(*
Nazwa:			FB_2GripperScrewers
Opis:			Zakręcarki szczekowe
Wersja:			v2.91
Data:			2026-01-12
Autor:			DP
Urzadzenia:		Serwo podnośnika, Serwo zakręcania
Ostatnie zmiany:
	- 2026-01-12 [DP] Wejście pod pozycje szukania gwintu
	- 2025-09-04 [DP] EventLog-do sprawdzenia->wywołać błędy , Estop ErrHan
	- 2025-07-09 [DP] wysokosc narzedi
	- 2025-07-08 [DP] tonError bo kasuje mcStop, tool height do błędu, opis, Resseting, Homing false w Manual
	- 2025-05-15 [DP] Zmiana errlowscrewing na -25
	- 2025-04-18 [DP] Zmiana limitu na 0.1 fullscr
	- 2025-03-31 [DP] Case 10 cofanie
	- 2025-03-31 [DP] Zmiana limitu lrPackageTurnoversToFullScrewed 0.3
	- 2025-01-17 [DP] TorqueCV 
	- 2024-12-13 [DP] Zmiany dla glowicy zasysajcej na sloiki, przejcie do pushing itd
	- 2024-12-12 [DP] Zmiana szukania gwintu
	- 2024-12-11 [DP] Skaling czuj. wysokości
	- 2024-11-26 [DP] Gear Vel sloiki
	- 2024-10-25 [DP] Zmiany torque
	- 2024-08-29 [DP] Wbijak
	- 2024-03-18 [DP] Zmiana symulacji
	- 2024-03-06 [DP] Aktualizacja instrukcji
	- 2024-02-27 [DP] Height Vel z 0 na zadaną w ressetingu, opis problemów
	- 2023-11-24 [DP] Pop. uwag dodatkowych opcji, tryb momentowy - opis
	- 2023-11-10 [DP] Akt. instrukcji, szukanie z UJL
	- 2023-03-25 [DP] przyśpieszenie screwera na stałe, zmiana instrukcji konfiguracji, skrocona czasowka griper
	- 2023-03-21 [DP] dodana ScrewerSet2
	- 2023-02-22 [DP] poprawa w GearRatio
	- 2023-02-21 [DP] Acc, Dec, Jerk i Prędkości Liftera zmniejszone 2x przez inny montaż,
				EStop w StateError, zmiana przekadni obrotu, CycleDone jak SetTorque=0,
	- 2023-02-14 [DP] Zmiana instrukcji konfiguracji
	- 2023-02-14 [DP] Wersja z LU208 z aktualizacjami z XTSa (gearing przy zakręcaniu i szukanie gwintu)
	
Konfiguracja:

Parametryzacja bloczka:
	- ustawić wysokości narzędzi, potrzebne do kolizji
	- ustawić wartość minimalną, od aktualnej wysokości zakręcarki
	

Czujnik wysokości:
	- Najlepiej przeskalować do na wejście tak, żeby pokazywał ugięcie sprężyny od transportera czyli 0mm-nieugięta
	14mm - ugięta maksymalnie (P10_GripperScrewer.IlrGripperScrewer1HeightCV:=-0.0023*(iIABPneumaticEB5AnalogueInput1)+52.006 + 1.83);

Szukanie gwintu z czujnikiem wysokości:
Włączone szukanie gwintu w pozycji dociskania i z czujnikiem wysokości, należy ustawić duży kąt obrotu (maxymalny dla szukania gwintu)
	1. Start obrotu z prędkością zadaną zakręcania, zapisywanie wartości max i min ugięcia sprężyny
	2. Szukanie 1 uskoku po 100st. o 0,5mm od wartości max ugięcia, jeżeli krotność gwintu 1x to przejście do punktu 4
	3. Szukanie 2 uskoku po 100st. jeżeli znaleziono pierwszy o 0,5mm od wartości max ugięcia
	4. Przejazd o 30,60,90st. dalej, zależnie od krotności
	5. Przejście do pozycji zakręcania lub dociskania zależnie od nastaw
	
	
Oś Obrótu (AM8031-0C20-0000): 

	Drive:
	- LU207,UBL50 - Nowa zębatka ma 32 na 48 zęby 240:360
	- ustawić driva na 'Rotatory' 360 st. i gear ratio 240:360, 240 st. na obr.
	- Invert Nc-Enc i Nc-Drive włączone
	- włączyć w drivie Scaling->Modulo data storage source - Feeback 1
	- ustawić drive Scaling->position offset setting 0 stopni na odpowiedniej pozycji na enkoderze
	- wgrać z drive Save NC parameters
	- w drivie jeszcze raz ustawić parametr Following error window 359?	
	- ustawic regulator Position mode na Kv na 10, Kp na 0.2, Tn na 0.002 
	- ustawić Acceleration Feed forward  K = 1 i wpisać inercje w Vel contr.->Vel. calc->0.001 kg m^2 oraz Mode->Basic_for_know_interia
	- ustawić w parametrach Configured channel peak current na 5A
	- ustawić w parametrach 0x6072 Bipolar torque/force limit value na 500%
	- ustawić w parametrach 0x60E0 Positive torque/force limit value na 500%
	- ustawić w parametrach 0x60E1 Negative torque/force limit value na 500%
	- dodać parametry Bipolar torque/Force limit w Process data/Outputs i polinkować ze zmienną
	- dodać parametr Positon control proportional gain Process data/Outputs i polinkować ze zmienną
	NC:
	- Ustawić Maximum Velocity na 13397.8, Reference Velocity na 14737.5, Max Acc i Dec na 300000.0
	- Default Acc i Dec na 20096.7, jerk na 60290.0
	- wyłączyć Limity Switche
	- wyłączyć wszystkie opcje Monitoringu

	Opcja trybu momentowego osi zakręcania (tylko od wersji driva 104)
	Drvie:
	- Na jednym drivie nie może być razem obrót 1 i obrót 2
	- W drivie (kanał) osi obrotu Advanced->Slots settings zaznaczyć 'I know what I do'
	i ustawiąc VelocityControlSlot na VelocityControl2, w tym momencie w IO powinny pojawić się 
	nowe wejścia,wyjścia VelocityControl2
	- W drivie Advanced->Process data rozwinąć 'Ch A Modes of operation' i ustawić '..mode_CST (10)'
	w Virual operation mode 0 
	- W parametr list powinien być parametr 0x60CA Ch a Torque limitation option code -> ustwić na
	TorqueMightBeReducedToZero, jeżeli nie ma to znaczy że trzeba zaktualizować driva lub dodać parametry ręcznie
	NC:
	- W NC w Drive->Zakładka Time Comensation-> Parametr Time Compensation Mode Drive -> 'ON(with velocity)'
	- W NC w Enc->Zakładka Time Comensation-> Parametr Time Compensation Mode Drive -> 'ON(with velocity)'
	
Oś podnoszenia (AM8032-0E21-0000):
	Drive:
	- ustawić driva na 'Linerary' 10mm i gear ratio 1:1, 10mm na obr.
	- Invert Nc-Enc i Nc-Drive włączone
	- ustawic regulator Position mode na Kv na 1, Kp na 0.2, Tn na 0.002 
	- ustawić Feed forward acceleration K = 1 i wpisać inercje w Vel contr.->Cel. calc->0 kg m^2
	NC:
	- Ustawić Maximum Velocity na 1094
	- Default Acc i Dec na 100000, jerk na 500000
	- ustawić Limit Swtiche
	- ustawić ManualVelocity (Slow) na 30 ze względu na Jog i bazowanie

Info: 
	- możliwość pracy 1 lub 2
	- możliwość pracy bez kręcenia jeżeli ustawi się prędkość 0
	- możliwosć dodatkowego chwytania przed zakręcaniem
	- step mode dla wizualizacji
	- rozróżnienie warningów

Tryb momementowy:
lrPackageTurnoversToFullScrewed - Ilośc obrotów do zakręcenia
iScrewer1SetTorque - Zadany moment w % (Przeliczany z Nm z wizualizacji)
lrScrewerSpeed - Prędkość zakręcania w st/s (Przeliczany z rpm z wizualziacji)
1. Start											Rozpędzanie,	Torque 5000 (Max) [%], 				TorqueRamp 4000 [%/s], VelocityLimitLow -5000 (Max) [st./s]
2. ActPos>lrPackageTurnoversToFullScrewed*360.0/7	Hamowanie,		Torque -9 [%],						TorqueRamp 1500 [%/s], VelocityLimitLow -4000 (Max) [st./s]
3. ActPos>lrPackageTurnoversToFullScrewed*360.0/6	Dokręcanie,		Torque iScrewer1SetTorque [%],		TorqueRamp 4000 [%/s], VelocityLimitLow lrScrewerSpeed (Max) [st./s]



Jak naprawić:
A. Zakręcarka nie wykonuje ruchu w trybie momentowym, jedna działa , druga nie - sprawdzić czy bloczek MC_Torque wykonuje ruchu,
jeżeli nie to wyłączyć VelocityControl2, włączyć bez '2' i ponownie włączyć '2', potem aktywacja
B. 
*)

FUNCTION_BLOCK FB_2GripperScrewers
VAR_INPUT
	bEnable1							:BOOL;		//Zezwolenie na pracę 1
	bEnable2							:BOOL;		//Zezwolenie na pracę 2
	bEstop								:BOOL;		//Stop awaryjny nieaktywny
	bRun1								:BOOL;		//Rozkaz zakręcania zakręcarki 1
	bRun2								:BOOL;		//Rozkaz zakręcania zakręcarki 2
	bSimulation							:BOOL;		//Włączona symulacja, skracanie czasu przerywania jak nie ma butelki
	bHoming								:BOOL;		//Zezwolenie na wykonanie bazowania i pozycjonowania zakręcarki
	bHeightSet							:BOOL;		//Ustaw wysokość
	bIgnoreError						:BOOL;		//Ignorowania błędów cyklu pracy
	bScrewer1SetPositionOffset			:BOOL;		//Ustaw offset obrotu zakręcarki 1
	bScrewer2SetPositionOffset			:BOOL;		//Ustaw offset obrotu zakręcarki 2
	iScrewer1AddTorque					:UINT;
	iScrewer2AddTorque					:UINT;
	bReset								:BOOL;		//Reset błędu, jeśli w stanie "eError
	iTool								:INT;		// Wybór narzędzia (1-5), opisy w tablicy AsGripperScrewerTool	
	bOptionOpenedGripperWhenFindingScrew:BOOL;		//OPCJA. Otwarty chwytak przy szukaniu gwintu
	bOptionScrewingBackwardsInPushingPosition:BOOL;	//OPCJA. Obrót do tyłu w pozycji dociskania
	bOptionCapPushingWithoutScrewing	:BOOL;		//OPCJA. Tylko wbijanie bez zakręcania
	bOptionCapPositioning				:BOOL;		//OPCJA. Dodatkowe zamknięcie chwytakiem przed zakręceniem (do testów)
	bOptionFindScrewInScrewingPosition	:BOOL;		//OPCJA. Szukaj początku gwintu nakrętki i opakowania. Zakręcarka napjpierw obraca się w lewo, a po znalezienu gwintu przystepuje do zakręcania w pozycji zakręcania
	bOptionFindScrewInPushingPosition	:BOOL;		//OPCJA. Szukaj początku gwintu nakrętki i opakowania. Zakręcarka napjpierw obraca się w lewo, a po znalezienu gwintu przystepuje do zakręcania w pozycsji docisku
	bOptionFindScrewWithHeightSensor	:BOOL;		//OPCJA. Szukanie gwintu z czujnikiem wysokości
	bOptionFindScrewRotateFromPushingToScrewingSensor	:BOOL;		//OPCJA. Obrót od pozycji docisku do zakręcania
	bOptionMomentaryMode				:BOOL;		//OPCJA. Tryb momentowy zakręcania
	lrPackageTurnoversToFullScrewed		:LREAL;		//Obroty do pełnego zakręcenia
	lrPackageThreadPitch				:LREAL;		//Skok gwintu
	lrPackageThreadTimes				:LREAL;		//Krotność gwintu
	lrHeightReadyPosition				:LREAL;		//Wysokość zadana w stanie gotowości od płyty[mm]
	lrHeightPushingPosition				:LREAL;		//Wysokość zadana przy wciskaniu nakrętki od płyty[mm]
	lrHeightEndScrewingPosition			:LREAL;		//Wysokość zadana przy zakręcaniu nakrętki od płyty [mm]
	lrHeightFindScrewPosition			:LREAL;		//Pozycja szukania gwintu [mm]
	lrHeightScrewingDistanceSpeed		:REAL;		//Prędkość obniżania podczas zakręcania
	lrHeightActualPosition				:LREAL;		//Aktualna pozycja podnośnika
	lrSpringHeightCV					:LREAL;		//Czujnik ugięcia sprężyny (przeskalować na 0-14mm (14mm-maksymalnie ugięta)
	lrHeightActualTorque				:LREAL;		//Aktualny moment [%]
	rActualMotor1Temperature			:REAL;		//Aktualna temperatura silnika 1
	rActualMotor2Temperature			:REAL;		//Aktualna temperatura silnika 2
	iHeightSetTorque					:INT;		//Zadany moment dociskania [%]
	iScrewer1SetTorque					:INT;		//Zadany moment dokręcania [%]
	iScrewer2SetTorque					:INT;		//Zadany moment dokręcania [%]
	iScrewTightTime						:INT;		//Czas przytrzymania po uzyskaniu momentu [ms] 
	lrScrewer1ActualTorque				:LREAL;		//Aktualny moment [%]
	lrScrewer2ActualTorque				:LREAL;		//Aktualny moment [%]
	lrHeightAcceleration				:LREAL;		//Przyspieszenie podnosnika zakręcarki
	lrHeightDeceleration				:LREAL;		//Opóźnienie podnośnika zakręcarki
	lrHeightSpeed						:LREAL;		//Prędkość podnośnika zakręcarki
	lrScrewer1ActualPosition			:LREAL;	
	lrScrewer2ActualPosition			:LREAL;	
	lrScrewerAcceleration				:LREAL;		//Przyspieszenie zakręcania
	lrScrewerDeceleration				:LREAL;		//Opóźnienie zakręcania
	lrScrewerSpeed						:LREAL;		//Prędkość zakręcania
	lrScrewer1PosDiff					:LREAL;		//ScrewingAxisRef.NcToPlc.PosDiff
	lrScrewer2PosDiff					:LREAL;		//ScrewingAxisRef.NcToPlc.PosDiff
	lrFindigScrewDegree					:LREAL;		//Kąt wycofania zakręcarki przy szukaniu gwintu
	bManualMovement						:BOOL;		//Zezwolenie na ruchy ręcznę
	lrManualOverride					:LREAL;		//Procentowa redukcja prędkości wszystkich serw (Tylko w trybie manualnym)
                                	
	lrMaxHeightPosition:LREAL;				//Wysokość maksymalna zakręcarki 
	lrMinHeightPosition:LREAL;				//Wysokość minimalna zakręcarki 
	lrMaxScrewerSpeed	:LREAL;				//Maksymalna prędkość zakręcania

	//StepMode
	bStepMode				: BOOL;		//Włączony tryb skokowy sterowania podnośnikami (tylko w serwisie)
	lrSetPosStepMode		: LREAL; 	//Ruch podnośnika o zadaną wartość w trybie krokowym (tylko w serwisie)
	
	_ALARMINFO_ :BOOL;
	iStationIndex:UDINT;					//Numer stacji 
	sStationName:WSTRING;					//Nazwa stacji
END_VAR

VAR_OUTPUT
	eState							: E_Station;				//Stan ogólny bloku
	eRunningState					: E_GripperScrewer; 		//Stan zakręcarki
	bError							: BOOL;						//Błąd stacji
	udiErrorID						: UDINT;					//Nr błędu zakręcarki
	sErrorDescription				: STRING(200);				//Opis błędu
	sErrorDescription2				: STRING(200);				//Opis błędu
	sErrorStationName				: STRING;					//Nazwa stacj
	udiStationID					: UDINT;				// Nr stacji
	
	udiHeightServoErrorNr			: UDINT;					//Nr błędu serwo podnośnika
	udiScrewing1ServoErrorNr		: UDINT;					//Nr błędu serwo zakręcarki 1
	udiScrewing2ServoErrorNr		: UDINT;					//Nr błędu serwo zakręcarki 2
	bGripper1Actuator				: BOOL;						//Siłownik chwytaka
	bGripper2Actuator				: BOOL;						//Siłownik chwytaka
	uiScrewing1TorqueControl		: UINT;						//Kontola momentu zakręcania	
	uiScrewing2TorqueControl		: UINT;						//Kontola momentu zakręcania	
	rScrewing1ProportionalGain		: UINT;						//Kontola Kp
	rScrewing2ProportionalGain		: UINT;						//Kontola Kp	
	lrScrewer1TorqueCV				: LREAL;					//Wartość osiągniętego momentu dokręcenia [nM]
	lrScrewer2TorqueCV				: LREAL;					//Wartość osiągniętego momentu dokręcenia [nM]
	uiHeightTorqueControl			: UINT						:= 6000;
	sWarningDescription				: STRING;
	bWarning1						: BOOL;
	bWarning1A						: BOOL;	
	bWarning1B						: BOOL;	
	bWarning1C						: BOOL;	
	bWarning1D						: BOOL;	
	bWarning1E						: BOOL;	{warning'dorobic ostrzezenie szukania gwintu}
	bWarning2						: BOOL;
	bWarning2A						: BOOL;	
	bWarning2B						: BOOL;	
	bWarning2C						: BOOL;	
	bWarning2D						: BOOL;	
	bWarning2E						: BOOL;	
	udiWarningID					: UDINT;
	tCycleTime						: TIME;	
	bHomingDone						: BOOL;						//Wymagane ponowne bazowanie (blad podczas bazowania lub stop awaryjny)
	bCycleDone1						: BOOL;
	bCycleNotDone1					: BOOL;		
	bCycleDone2						: BOOL;
	bCycleNotDone2					: BOOL;		
	bAdjustingTorqueDone			: BOOL;
	iAdjustingTorque				: INT;
	lrAdjustingMaxTorque			: LREAL;
	AsToolDescription				: ARRAY [0..10] OF STRING;	// Opis narzędzi, 1 - Opis narzędzia nr 1, 2 - Opis narzędzia nr 2
	sTool							: STRING;
	iToolHeight						: INT;	//Wysokość narzędzia od dolnej metalowej częsci dwuszczekowego
END_VAR

VAR_IN_OUT
	bManualHeightUp					:BOOL;			//Ruch ręczny podnośnikiem stacji w górę
	bManualHeightDown				:BOOL;			//Ruch ręczny podnośnikiem stacji w dół
	bManualScrew1Clockwise			:BOOL;			//Ruch ręczny zakręcarką w kierunku wskazówek zegara;
	bManualScrew1CClockwise			:BOOL;			//Ruch ręczny zakręcarką w kierunku przeciwnym do wskazówek zegara;
	bManualScrew2Clockwise			:BOOL;			//Ruch ręczny zakręcarką w kierunku wskazówek zegara;
	bManualScrew2CClockwise			:BOOL;			//Ruch ręczny zakręcarką w kierunku przeciwnym do wskazówek zegara;
	bManualGripper1					:BOOL;			//Ruch zamknięcie chwytaka nakrętek
	bManualGripper2					:BOOL;			//Ruch zamknięcie chwytaka nakrętek
	HeightAxisRef					:AXIS_REF;		//Struktura sterowania NC dla serwa podnoszenia zakręcarki
	Screwing1AxisRef				:AXIS_REF;		//Struktura sterowania NC dla serwa zakręcania
	Screwing2AxisRef				:AXIS_REF;		//Struktura sterowania NC dla serwa zakręcania	
	bFindScrewAdjustSensorHeight	:BOOL;			//Włacz szukanie MIN i MAX jeżeli jest opcja z czujnikie wysokości
	bAdjustingTorque				:BOOL;			//Dobieranie momentu
	lrAdjustingSetTorque			:LREAL;	
END_VAR

VAR
	bScrew1Found					: BOOL; 						// Zakręcarka znalazła początek gwintu
	bScrew2Found					: BOOL; 						// Zakręcarka znalazła początek gwintu	
	tonTightScrewing1Timer			: TON; 							// Timer potwierdzenia dokręcenia nakrętki
	tonTightScrewing2Timer			: TON; 							// Timer potwierdzenia dokręcenia nakrętki
	tonTightScrewing1TimerAndOpenedGripper	: TON; 					// Timer potwierdzenia dokręcenia nakrętki
	tonTightScrewing2TimerAndOpenedGripper	: TON; 					// Timer potwierdzenia dokręcenia nakrętki	
	tonMomentaryScrewing1Timer		: TON; 							// Timer potwierdzenia dokręcenia nakrętki
	tonMomentaryScrewing2Timer		: TON; 							// Timer potwierdzenia dokręcenia nakrętki

	bScrewed1					: BOOL; 						// Nakrętka zakręcona
	bScrewed2					: BOOL; 						// Nakrętka zakręcona
	tonTooLongScrewing1			: TON;							// Błąd zbyt długiego zakręcania
	tonTooLongScrewing2			: TON; 							// Błąd zbyt długiego zakręcania	
	tTooLongScrewing1			: TIME;							// Czas  zbyt długiego zakręcania
	tTooLongScrewing2			: TIME; 						// Czas  zbyt długiego zakręcania		
	tonGripper1ReliseDelay		: TON;							// Time Opóźniajacy ruch w górę po zakręceniu, pozwalajac na otwarcie chwytaka
	tonGripper2ReliseDelay		: TON;							// Time Opóźniajacy ruch w górę po zakręceniu, pozwalajac na otwarcie chwytaka
	tonGripper1ReliseDelay2		: TON;							// Time Opóźniajacy ruch w górę po zakręceniu, pozwalajac na otwarcie chwytaka
	tonGripper2ReliseDelay2		: TON;							// Time Opóźniajacy ruch w górę po zakręceniu, pozwalajac na otwarcie chwytaka

	mcScrewer1ManualMove		: MC_JOG; 						// Blok obrotu ręcznego zakręcarką
	mcScrewer2ManualMove		: MC_JOG; 						// Blok obrotu ręcznego zakręcarką
	mcScrewer1Stop				: MC_Stop;						// Trwałe zatrzymywanie Serwo
	mcScrewer2Stop				: MC_Stop;						// Trwałe zatrzymywanie Serwo
	mcScrewer1MoveVelocity		: MC_MoveVelocity;				// Ruch prędkościowy
	mcScrewer2MoveVelocity		: MC_MoveVelocity;				// Ruch prędkościowy
	mcScrewer1MoveVelocity2		: MC_MoveVelocity;				// Ruch prędkościowy
	mcScrewer2MoveVelocity2		: MC_MoveVelocity;				// Ruch prędkościowy
	mcScrewer1MoveVelocity3		: MC_MoveVelocity;				// Ruch prędkościowy
	mcScrewer2MoveVelocity3		: MC_MoveVelocity;				// Ruch prędkościowy	
	mcScrewer1MoveRelative		: MC_MoveRelative; 				// Ruch relatywny zakręcarki
	mcScrewer2MoveRelative		: MC_MoveRelative; 				// Ruch relatywny zakręcarki
	mcScrewer1MoveAbsolute		: MC_MoveAbsolute; 				// Ruch absolutny zakręcarki
	mcScrewer2MoveAbsolute		: MC_MoveAbsolute; 				// Ruch absolutny zakręcarki
	fbScrewer1SetPositionOffset	: FB_CoEAX8000SetPositionOffset;// Ustawianie pozycji obrotu 
	fbScrewer2SetPositionOffset	: FB_CoEAX8000SetPositionOffset;// Ustawianie pozycji obrotu 
	mcScrewer1TorqueControl		: MC_TorqueControl;
	mcScrewer2TorqueControl		: MC_TorqueControl;
	
	mcScrewing1Power			: MC_Power;			 			// Zasilanie napędu zakręcarki
	mcScrewing2Power			: MC_Power;			 			// Zasilanie napędu zakręcarki
	bScrewer1ServoPower			: BOOL; 						// Zmienna sterujaca zasilaniem serwo Zakręcarki
	bScrewer2ServoPower			: BOOL; 						// Zmienna sterujaca zasilaniem serwo Zakręcarki
	fbScrewer1HardReset			: FB_SoEReset; 					// Blok twardego resetu serwa zakręcania
	fbScrewer2HardReset			: FB_SoEReset; 					// Blok twardego resetu serwa zakręcania
	mcScrewer1SoftReset			: MC_Reset; 					// blok łagodnego resetu serwa zakręcarki
	mcScrewer2SoftReset			: MC_Reset; 					// blok łagodnego resetu serwa zakręcarki
	
	mcHeightManualMove			: MC_JOG; 						// Blok sterowania ręcznego wysokością
	mcHeightStop				: MC_STOP; 						// Trwałe Zatrzymywanie ruchu podnośnika zakręcarki
	mcHeightMoveAbsolute		: MC_MoveAbsolute;				// Blok sterowania wysokością	
	mcHeightPower				: MC_POWER; 					// Uruchomienie zasilania serwa podnosnika zakręcarki
	bHeightServoPower			: BOOL; 						// Zmienna sterowania zasilaniem serwo
	fbHeightHardReset			: FB_SoEReset; 					// Blok Twardego resetu serwa podnośnika zakręcarki
	mcHeightSoftReset			: MC_Reset; 					// Blok łagonego resetu podnośnika zakręcarki
	mcHeightGearInMultiMaster	: MC_GearInMultiMaster; 		// Blok sprzęgania podnoszenia z zakręcaniem
	mcHeightGearOut				: Mc_GearOut;					// Blok wysprzeglania podnoszenia z zakręcaniem

	(*Axis online*)
	fbHeight					: FB_McAxisOnlineAX8000;
	stHeight					: ST_McAxisOnline;
	fbScrewing1					: FB_McAxisOnlineAX8000;
	stScrewing1					: ST_McAxisOnline;
	fbScrewing2					: FB_McAxisOnlineAX8000;
	stScrewing2					: ST_McAxisOnline;
	
	(*Ostrzezenia,przerywanie*)
	tonTooLongFinding1			: TON; 							// Za długie szukanie gwintu
	tonTooLongFinding2			: TON; 							// Za długie szukanie gwintu
	tonPosDiff1Error			: TON;
	tonPosDiff2Error			: TON;
	tonPosTooLowWhenScrewing1	: TON;
	tonPosTooLowWhenScrewing2	: TON;
	
	(*Statistics*)
	tonCycleTimer				: TON;
	rtrigCycleTimerRead			: R_TRIG;

	lrStartPosition1			: LREAL;
	lrStartPosition2			: LREAL;
	tonMaxHeight				: TON;

	tonGripper1Delay			: TON;
	tonGripper2Delay			: TON;
	
	eLastState					: E_Station;			// Stan ogólny bloku
	eLastRunningState			: E_GripperScrewer;		// Stan podbloku
	eLastStateTemp				: E_Station;			// Stan ogólny bloku
	eLastRunningStateTemp		: E_GripperScrewer;		// Stan podbloku

	bStateError: BOOL;
	bHeighSetNotDone: BOOL;
	
	(*Szukanie momentu*)
	nCaseAdjustingTorque					: INT;
	tonAdjustingTightScrewingTimer			: TON;
	tonAdjustingGripperClose				: TON;
	uiAdjustingScrewerTorqueControl			: UINT;
	bAdjustingScrewed						: BOOL;
	tonAdjustingCase40						: TON;
	bAdjustingSetTorqueAchieved				: BOOL;
	bAdjustingTorqueTooHigh					: BOOL;
	bAdjustingTorqueTooLow					: BOOL;
	lrMotorNominalTorque					: LREAL;
	lrScrewerActualTorqueNm					: LREAL;
	
	tonFindingScrew						: TON;
	tonScrew1Found						: TON;
	tonScrew2Found						: TON;
	tonDelayServoOn						: TON;

	bPreparingToDisable					: BOOL;
	bHeightGearingWithScrewer			: BOOL;
	iStoppingCase						: INT;
	iScrewingCase						: INT;
	iScrewing2Case						: INT;
	
	(*Bledy, Resetowanie*)
	tonResetting						: TON;
	tonEstop							: TON;
	tonError							: TON;	
	rtResetCommands						: R_TRIG;
	tonActualMotor1TemperatureTooHigh	: TON;
	tonActualMotor2TemperatureTooHigh	: TON;
	iErrorResseting3					: INT;
	iTestError3							: INT;
	iTestError4							: INT;
	
	(*Metoda*)
	mcMoveAbsolute						: MC_MoveAbsolute; 				// Ruch absolutny
	iMStep								: INT;							// Do testów
	bPrepareToReadyTest					: BOOL;							// Do testów	

	(*Bazowanie*)
	iHomingCase							: INT;
	iPreparingToReadyCase				: INT;
	
	(*Czytanie momentu*)
	rtRun1								: R_TRIG;
	rtRun2								: R_TRIG;

	(*Step Mode*)
	rtStepModeUp						: R_TRIG;
	rtStepModeDown						: R_TRIG;
	lrStepModeHeightMotorSV				: LREAL;
	bStepModeMoving						: BOOL;
	tofStepModeMoving					: TOF;	
	
	(*Running*)
	iGoingUpCase						: INT;
	iToPushingPositionCase				: INT;
	tonDelayBeforeResetLag				: TON;
	lrGearRatio1						: LREAL;
	lrGearRatio2						: LREAL;
	lrSf1								: LREAL;	
	lrSf2								: LREAL;
	lrDivider							: LREAL;	
	
	(*Dodatkowe chwytanie przed zakreceniem*)
	iCloseGripperBeforeScrewingCASE		: INT;
	
	(*Bez zakręcania*)
	tonHoldingTimer						: TON;
	
	(*Aborting*)
	iAbortingCASE						: INT;
	
	(*Szukanie gwintu*)
	iFindingScrewCASE							: INT;
	lrScrewer1MaxTorqueWhenFindingScrew			: LREAL; //OPCJA 1
	lrScrewer2MaxTorqueWhenFindingScrew			: LREAL; //OPCJA 1	
	lrScrewerMinTorqueWhenFindingScrew			: LREAL; //OPCJA 1
	lrScrewerMaxSensorHeightWhenFindingScrew	: LREAL:= -100000; //OPCJA 2
	lrScrewerMinSensorHeightWhenFindingScrew	: LREAL:= 0; //OPCJA 2
	bScrew1MinFound								: BOOL;
	bScrew2MinFound								: BOOL;
	lrStartPosition1FindingScrew				: LREAL;
	lrStartPosition2FindingScrew				: LREAL;
	lrFindingScrewPositionDelay					: LREAL;	
	tonFindingScrewDelay						: TON;
	iFindScrewAdjustSensorHeight				: INT;
	
	(*Symulacja*)
	tonSimulationScrewing1						: TON;
	tonSimulationScrewing2						: TON;	
	
	(*inne*)
	iTestResetting: INT;
	iCountAborting: INT;
	bTest2:BOOL;
	lrScrewerOffsetSensorHeightWhenFindingScrew: LREAL;
	bTest: BOOL;
	iTesty: INT;
	tonTesty1: TON;
	tonTesty2: TON;	
	
	//Zmienne od EVENTLOGGER
	bAlarmInit 						: BOOL := TRUE; 
	nAlarmNumerator					: INT;
	arfbAlarm						: ARRAY[0..19] OF  FB_TcAlarm;		//Tablica bloczków błędów
	fbSourceInfo 					: FB_TcSourceInfo;
	iSourceInfo						: I_TcSourceInfo;
	sAlarmTest						: STRING;
	//Koniec zmiennych od EVENTLOGGER
	
END_VAR

IF bPrepareToReadyTest THEN
	IF	M_PrepareToReady(	AxisRef			:=  Screwing1AxisRef,			
                   			iGripperArms	:=	2
						)	
	THEN
		bPrepareToReadyTest := FALSE;
	END_IF			
				   
END_IF  

//Wywołanie AXIS Online
(*fbHeight	(stMcAxisOnline:= stHeight,		Axis:= HeightAxisRef);
fbHeight	(stMcAxisOnline:= stHeight,		Axis:= HeightAxisRef);
fbScrewing1	(stMcAxisOnline:= stScrewing1,	Axis:= Screwing1AxisRef);
fbScrewing1	(stMcAxisOnline:= stScrewing1,	Axis:= Screwing1AxisRef);
fbScrewing2	(stMcAxisOnline:= stScrewing2,	Axis:= Screwing2AxisRef);
fbScrewing2	(stMcAxisOnline:= stScrewing2,	Axis:= Screwing2AxisRef);
*)
//Parametryzacja
bHeightGearingWithScrewer := TRUE;

Tools();
ErrorHandling();
Control();
Limits();
AdjustingTorque();
HeightControlBlocks();
TorqueControl();
Screwer1ControlBlocks();
Screwer2ControlBlocks();
Simulation();
ReadScrewingTorque();
Statistics();
Warnings();
aStationID();
aTesty();
(*Zapisywanie ostatniego stanu*)
IF eLastStateTemp<>eState THEN
	eLastState := eLastStateTemp;
END_IF
eLastStateTemp := eState;
IF eLastRunningStateTemp<>eRunningState THEN
	eLastRunningState := eLastRunningStateTemp;
END_IF
eLastRunningStateTemp := eRunningState;
(*Koniec Zapisywanie ostatniego stanu*)


(*Dodatkowe zabezpieczenie przed uderzeniem w chwytak*)
IF mcHeightMoveAbsolute.Execute AND (mcHeightMoveAbsolute.Position-iToolHeight)<=lrMinHeightPosition THEN
	mcHeightMoveAbsolute.Execute:=FALSE;
END_IF
	
IF mcHeightMoveAbsolute.Error THEN
	mcHeightMoveAbsolute.Execute:=FALSE;
END_IF

IF mcScrewer1MoveVelocity.Error THEN
	mcScrewer1MoveVelocity.Execute:=FALSE;
END_IF	
(*Koniec dodatkowe zabezpieczenie przed uderzeniem w chwytak*)


(*Zabezpieczenie przed kolizją stacji poprzez ruch podnośnika*)	
IF bManualHeightDown AND (HeightAxisRef.NcToPlc.ActPos-iToolHeight)<=lrMinHeightPosition AND NOT bHoming AND NOT bHeightSet THEN
	bManualHeightDown:=FALSE;
END_IF	

IF bManualHeightUp AND (HeightAxisRef.NcToPlc.ActPos)>=lrMaxHeightPosition AND NOT bHoming AND NOT bHeightSet THEN
	bManualHeightUp:=FALSE;
END_IF	
(*Koniec zabezpieczenia przed kolizją stacji poprzez ruch podnośnika*)

ACTION AdjustingTorque:
(*

bAdjustingTorque;								// Wlączenie szukania 
lrAdjustingSetTorque;							// Szukany moment [Nm]
uiAdjustingScrewerTorqueControl; 				// Badanie tym momentem, zwiekszanie o ileś
lrMotorNominalTorque					:=	3.192; 		

tonAdjustingGripperClose		(IN:=	bGripper1Actuator, 																		PT:=T#200MS);
tonAdjustingTightScrewingTimer	(IN:=	nCaseAdjustingTorque = 30 AND (lrScrewer1ActualTorque>=uiAdjustingScrewerTorqueControl),	PT:=T#1000MS);
tonAdjustingCase40				(IN:=	nCaseAdjustingTorque=40,																PT:=T#200MS);

CASE nCaseAdjustingTorque OF
	
	0: //Włączanie
		IF bAdjustingTorque AND NOT bAdjustingTorqueDone THEN
			//Kasowanie zmiennych
			lrStartPosition1				:=	0;
			uiAdjustingScrewerTorqueControl	:=	0;
			iAdjustingTorque				:=  0;
			lrAdjustingMaxTorque			:= 	0;
			bAdjustingTorqueTooHigh			:=	FALSE;
			bAdjustingTorqueTooLow			:=	FALSE;
			nCaseAdjustingTorque			:=	10;
			mcScrewer1MoveVelocity.Execute	:=	FALSE;
		END_IF
		
	10: //Zamykanie chwytaka
		bGripper1Actuator					:=	TRUE;
		IF tonAdjustingGripperClose.Q THEN
			nCaseAdjustingTorque			:=	20;
		END_IF
		
	20:	//Ustawienie dużego momentu na początek ruchu
		uiScrewing1TorqueControl				:=  6000;
		lrStartPosition1						:=	Screwing1AxisRef.NcToPlc.ActPos;		

		IF  bAdjustingTorqueTooLow	THEN
			bAdjustingTorqueTooLow				:= FALSE;
			uiAdjustingScrewerTorqueControl		:=  uiAdjustingScrewerTorqueControl + 1;
		ELSIF bAdjustingTorqueTooHigh	THEN
			bAdjustingTorqueTooHigh				:= FALSE;
			IF uiAdjustingScrewerTorqueControl	>	0 THEN
			uiAdjustingScrewerTorqueControl		:=  uiAdjustingScrewerTorqueControl - 1;
			END_IF
		END_IF
		nCaseAdjustingTorque				:=	30;
		
	30:	 //Zakręcanie

		//Zacznij zakręcać
		lrScrewerAcceleration				:=	26000;
		lrScrewerDeceleration				:=	26000;
		mcScrewer1MoveVelocity.Direction		:=	MC_Positive_Direction;
		mcScrewer1MoveVelocity.Velocity		:=	5000;
		mcScrewer1MoveVelocity.Execute		:=	TRUE;
		
		//Zwiększanie momentu na początek ruchu
		IF ABS(ABS(lrStartPosition1)-ABS(Screwing1AxisRef.NcToPlc.ActPos))>15 OR ABS(Screwing1AxisRef.NcToPlc.PosDiff)>15  THEN 
			uiScrewing1TorqueControl			:=	(uiAdjustingScrewerTorqueControl+3)*10;
		ELSE
			uiScrewing1TorqueControl			:=	(uiAdjustingScrewerTorqueControl+3)*10+500;	
		END_IF
		
		IF tonAdjustingTightScrewingTimer.Q THEN //Jeżeli osiągnięty moment przez 200MS
			mcScrewer1MoveVelocity.Execute	:=	FALSE;
			mcScrewer1SoftReset				(Axis:=Screwing1AxisRef, Execute:= TRUE);
			iAdjustingTorque				:= UINT_TO_INT(uiScrewing1TorqueControl/10);
			uiScrewing1TorqueControl			:=	0;
			bAdjustingScrewed				:=	TRUE;		
		END_IF
			   
		IF mcScrewer1MoveVelocity.Execute = FALSE AND bAdjustingScrewed THEN
			nCaseAdjustingTorque			:=	40;
		
		END_IF	
		
	40:	//Czekanie po zakręceniu
		mcScrewer1SoftReset					(Axis:=Screwing1AxisRef, Execute:= FALSE);
		uiScrewing1TorqueControl				:=	0;
		lrStartPosition1						:=	0;
		lrAdjustingMaxTorque				:= 	0;
		bAdjustingScrewed					:=	FALSE;
		IF tonAdjustingCase40.Q THEN
			lrStartPosition1					:=	Screwing1AxisRef.NcToPlc.ActPos;	
			uiScrewing1TorqueControl			:=	1;
			nCaseAdjustingTorque			:=	50;
		END_IF
		
	50: //Odkręcanie

		lrScrewerAcceleration				:=	20;
		lrScrewerDeceleration				:=	20;
		mcScrewer1MoveVelocity.Direction		:=	MC_Negative_Direction;
		mcScrewer1MoveVelocity.Velocity		:=	10;
		mcScrewer1MoveVelocity.Execute		:=	TRUE;
		uiScrewing1TorqueControl				:=	6000;
		
		//Szukanie największego momentu w Nm
		lrScrewerActualTorqueNm:=(ABS(lrScrewer1ActualTorque)/100.0)*lrMotorNominalTorque;
		IF lrScrewerActualTorqueNm	>=	lrAdjustingMaxTorque THEN
			lrAdjustingMaxTorque			:=	lrScrewerActualTorqueNm;
		END_IF
		
		//Jeżeli osiągnięty moment
		IF lrAdjustingMaxTorque>=lrAdjustingSetTorque - 0.1 AND lrAdjustingMaxTorque<=lrAdjustingSetTorque + 0.1 THEN
			bAdjustingSetTorqueAchieved 	:= TRUE;
		ELSE
			bAdjustingSetTorqueAchieved 	:= FALSE;
		END_IF
		
		
		//Odkręcone ale nie z zadanym momentem
		IF ABS(Screwing1AxisRef.NcToPlc.ActPos-lrStartPosition1) > 45 OR ABS(Screwing1AxisRef.NcToPlc.PosDiff) > 45  THEN
			mcScrewer1SoftReset				(Axis:=Screwing1AxisRef, Execute:= TRUE);
			mcScrewer1MoveVelocity.Execute	:=	FALSE;
			
			IF lrAdjustingMaxTorque >= lrAdjustingSetTorque + 0.1 THEN
				bAdjustingTorqueTooHigh		:= TRUE;
			ELSIF lrAdjustingMaxTorque <= lrAdjustingSetTorque - 0.1 THEN
				bAdjustingTorqueTooLow		:= TRUE;	
			END_IF				
			nCaseAdjustingTorque			:= 60;
			
		END_IF
		
		//Pozycja aktualna jest większa niż 1/4 obrotu
		IF bAdjustingSetTorqueAchieved AND ABS(Screwing1AxisRef.NcToPlc.ActPos-lrStartPosition1)>45 THEN
			mcScrewer1SoftReset				(Axis:=Screwing1AxisRef, Execute:= TRUE);
			mcScrewer1MoveVelocity.Execute	:=	FALSE;
			nCaseAdjustingTorque			:= 100;
		END_IF
		
		
	60: //Ponowne zwiększanie momentu
	
		mcScrewer1SoftReset					(Axis:=Screwing1AxisRef, Execute:= FALSE);
		bAdjustingSetTorqueAchieved 		:=	FALSE;
		nCaseAdjustingTorque				:= 20;	



		
	100: //Moment znaleziony
		
		iAdjustingTorque;
		bGripper1Actuator					:= FALSE;
		nCaseAdjustingTorque				:= 0;
		//bAdjustingTorque 					:= FALSE;
		mcScrewer1MoveVelocity.Direction		:=	MC_Positive_Direction;	
		bAdjustingTorqueDone				:= TRUE;
	
END_CASE

//Resetowanie gdy wyłączono w trakcie
IF nCaseAdjustingTorque > 0 AND NOT bAdjustingTorque THEN

		lrStartPosition1					:=	0;
		uiAdjustingScrewerTorqueControl	:=	0;
		iAdjustingTorque				:=  0;
		lrAdjustingMaxTorque			:= 	0;
		bAdjustingTorqueTooHigh			:=	FALSE;
		bAdjustingTorqueTooLow			:=	FALSE;
		bAdjustingTorqueDone			:= FALSE;
		mcScrewer1Stop.Execute			:=	TRUE;
		IF mcScrewer1Stop.Done THEN
					mcScrewer1Stop.Execute			:=	FALSE;
					nCaseAdjustingTorque			:=	0;
		END_IF
END_IF

//Kasowanie Done
IF NOT bAdjustingTorque THEN 
				bAdjustingTorqueDone			:= FALSE;
END_IF
*)
END_ACTION

ACTION aStationID:
udiStationID	:=	iStationIndex;
END_ACTION

ACTION aTesty:
mcHeightMoveAbsolute;
tonTesty1	(IN:=iTesty=30, PT:=T#100MS);
tonTesty2	(IN:=iTesty=60, PT:=T#1000MS);

CASE iTesty OF 
	
		0:
			;
			
		10: 
		
			mcHeightMoveAbsolute.Execute						:=	TRUE;
			mcHeightMoveAbsolute.Velocity						:=	lrHeightSpeed;
			mcHeightMoveAbsolute.Position						:=	300;
			IF mcHeightMoveAbsolute.Done THEN
				mcHeightMoveAbsolute.Execute					:= FALSE;
				iTesty	:=	iTesty	+	10;
			END_IF
			
		20:
			mcHeightMoveAbsolute.Execute						:=	TRUE;
			mcHeightMoveAbsolute.Velocity						:=	lrHeightSpeed;
			mcHeightMoveAbsolute.Position						:=	250;
			IF mcHeightMoveAbsolute.Done THEN
				mcHeightMoveAbsolute.Execute					:= FALSE;
				iTesty	:=	iTesty	+	10;
			END_IF
			
		30:
			IF tonTesty1.Q THEN
				iTesty	:=	iTesty	+	10;
			END_IF
		
		40:
		
			mcHeightMoveAbsolute.Execute						:=	TRUE;
			mcHeightMoveAbsolute.Velocity						:=	lrHeightSpeed;
			mcHeightMoveAbsolute.Position						:=	300;
			IF mcHeightMoveAbsolute.Done THEN
				mcHeightMoveAbsolute.Execute					:= FALSE;
				iTesty	:=	iTesty	+	10;
			END_IF

		50:
		
			mcHeightMoveAbsolute.Execute						:=	TRUE;
			mcHeightMoveAbsolute.Velocity						:=	lrHeightSpeed;
			mcHeightMoveAbsolute.Position						:=	200;
			IF mcHeightMoveAbsolute.Done THEN
				mcHeightMoveAbsolute.Execute					:= FALSE;
				iTesty	:=	iTesty	+	10;	
			END_IF
		60:
			IF tonTesty2.Q THEN
				iTesty	:=	iTesty	+	10;
			END_IF	
	
		70:	
			mcHeightMoveAbsolute.Execute						:=	TRUE;
			mcHeightMoveAbsolute.Velocity						:=	lrHeightSpeed;
			mcHeightMoveAbsolute.Position						:=	300;
			IF mcHeightMoveAbsolute.Done THEN
				mcHeightMoveAbsolute.Execute					:= FALSE;
				iTesty	:=	iTesty	+	10;
			END_IF
			
		80:
			;

END_CASE
END_ACTION

ACTION Control:
	(** TIMERY**)
	tonGripper1ReliseDelay	(IN:=	NOT bGripper1Actuator, 					PT:=T#70MS);	//bylo 50,140
	tonGripper2ReliseDelay	(IN:=	NOT bGripper2Actuator, 					PT:=T#70MS);	//bylo 50,140
 	tonGripper1ReliseDelay2	(IN:=	NOT bGripper1Actuator, 					PT:=T#80MS);	
	tonGripper2ReliseDelay2	(IN:=	NOT bGripper2Actuator, 					PT:=T#80MS);	
                                 	
	IF iTool = 4 THEN // tylko dla glowicy zasysajacej 400ms
		tonGripper1Delay		(IN:=	bGripper1Actuator, 						PT:=T#400MS);	
		tonGripper2Delay		(IN:=	bGripper2Actuator, 						PT:=T#400MS);	
    ELSE
		tonGripper1Delay		(IN:=	bGripper1Actuator, 						PT:=T#100MS);	//bylo 50  /// jednak 150
		tonGripper2Delay		(IN:=	bGripper2Actuator, 						PT:=T#100MS);	//bylo 50 /// a jednak 150	
	END_IF
                  																																								// Nie moze być 60 bo nalicza 60 i powyzej 360 sie przekręca																			
	tonTightScrewing1Timer	(IN:=		(eRunningState=E_GripperScrewer.eScrewing) AND 
									NOT tonTightScrewing1Timer.Q AND 
										(mcScrewer1MoveVelocity.Execute OR mcScrewer1MoveVelocity3.Execute) 		AND 
										(mcScrewer1MoveVelocity.InVelocity OR mcScrewer1MoveVelocity3.InVelocity)	AND 
										(
											Screwing1AxisRef.NcToPlc.ActVelo < 100 (*AND ABS(Screwing1AxisRef.NcToPlc.PosDiff)>60 *) OR
											iScrewer1SetTorque = 0 OR 
											tonSimulationScrewing1.Q
										)	
 										AND 
									NOT bScrewed1
										,PT:=INT_TO_TIME(iScrewTightTime));
	tonTightScrewing2Timer	(IN:=	(eRunningState=E_GripperScrewer.eScrewing) AND
									 NOT tonTightScrewing2Timer.Q AND 
										(mcScrewer2MoveVelocity.Execute OR mcScrewer2MoveVelocity3.Execute) 		AND 
										(mcScrewer2MoveVelocity.InVelocity OR mcScrewer2MoveVelocity3.InVelocity) 	AND 
										(
											Screwing2AxisRef.NcToPlc.ActVelo < 100 (*AND ABS(Screwing2AxisRef.NcToPlc.PosDiff)>60 *) OR 
											iScrewer2SetTorque = 0 OR 
											tonSimulationScrewing2.Q
										)
										AND 
									NOT bScrewed2
										,PT:=INT_TO_TIME(iScrewTightTime));
	
	tonTightScrewing1TimerAndOpenedGripper(IN:=bScrewed1,	PT:=T#140MS); //bylo 100
	tonTightScrewing2TimerAndOpenedGripper(IN:=bScrewed2,	PT:=T#140MS); //bylo 100

	tonMomentaryScrewing1Timer	(IN:=	(eRunningState=E_GripperScrewer.eScrewing)	AND NOT tonMomentaryScrewing1Timer.Q AND 
											mcScrewer1TorqueControl.Active 		AND 
											Screwing1AxisRef.NcToPlc.ActVelo < 100  AND NOT bScrewed1,
										PT:=INT_TO_TIME(iScrewTightTime+20));
	tonMomentaryScrewing2Timer	(IN:=	(eRunningState=E_GripperScrewer.eScrewing)	AND NOT tonMomentaryScrewing2Timer.Q AND 
											mcScrewer2TorqueControl.Active 		AND 
											Screwing2AxisRef.NcToPlc.ActVelo < 100  AND NOT bScrewed2,
										PT:=INT_TO_TIME(iScrewTightTime+20));
	
	tonHoldingTimer			(IN:=	(eRunningState=E_GripperScrewer.eHolding ),	PT:=INT_TO_TIME(iScrewTightTime));
                  	
	tonDelayServoOn			(IN:=	(eState = E_Station.ePreparingToReady), PT:=T#7S); //bylo 1,2s
	tonResetting			(IN:=	(eState = E_Station.eResetting), 		PT:=T#1000MS);
	
	rtResetCommands			(CLK:=	eState = E_Station.eReady (* OR *)		,Q=>); //Triger do resetu zmienych
	tonDelayBeforeResetLag 	(IN:=	iGoingUpCase=10, 				PT:=T#10MS);

	tonFindingScrewDelay 	(IN:=	iFindingScrewCASE = 50, 				PT:=T#0MS);
	tonEStop				(IN:=	bEstop,									PT:=T#2S);
	tonError				(IN:=	eState = E_Station.eError, 			PT:=T#1000MS);
	
	(*****Wyłączenie enable*****)
	IF NOT bEnable1 AND NOT bEnable2 AND NOT bError THEN
		IF eState <> E_Station.eDisabled AND eState <> E_Station.ePreparingToDisable AND eState <> E_Station.eAborting AND  eState <> E_Station.eAborted THEN
			eState 				:= E_Station.ePreparingToDisable; 
		END_IF	
	END_IF

	(*****Estop*****)
	IF NOT bEstop  THEN	
		IF eState <> E_Station.eAborted AND eState <> E_Station.eAborting AND eState <> E_Station.eDisabled THEN
				iAbortingCASE		:=	0;
				eState 				:=	E_Station.eAborting; 
		END_IF
	END_IF

	
	CASE eState OF
	/////////////////////////////	
		E_Station.eDisabled: 					// Stan nieaktywnosci (Stacja wyłączona) 
		
			IF bEnable1 OR bEnable2 THEN
				eState 				:= E_Station.ePreparingToReady; 
			END_IF 
			
    /////////////////////////////	    
		E_Station.eAborted: 					// Stan bezpiecznego zatrzymania (po Abortingu) 

			IF bEStop THEN
				eState 				:= E_Station.ePreparingToReady;
			END_IF
			
	/////////////////////////////	
		E_Station.eAborting:                 	// Stan bezpiecznego zatrzymywania (po EStopie)
		
			CASE iAbortingCASE OF   
				0: //Czyszczenie
					ResetCommands(); 
					iAbortingCASE	:=	iAbortingCASE	+	10;
//					iCountAborting	:=	iCountAborting	+	1;
				10: //Stop
					mcHeightPower.Override			:=	100;
					mcScrewing1Power.Override		:=	100;
					mcScrewing2Power.Override		:=	100;
		
					//F NOT mcHeightStop.Error AND NOT mcScrewer1Stop.Error AND NOT mcScrewer2Stop.Error THEN
					mcHeightStop.Execute			:=	TRUE;
					mcScrewer1Stop.Execute			:=	TRUE;
					mcScrewer2Stop.Execute			:=	TRUE;	
					iAbortingCASE					:=	iAbortingCASE	+	10;	
					//ELSE
				(*	mcHeightStop.Execute			:=	FALSE;
					mcScrewer1Stop.Execute			:=	FALSE;
					mcScrewer2Stop.Execute			:=	FALSE;
					bHeightServoPower				:=	FALSE;
					bScrewer1ServoPower				:=	FALSE;
					bScrewer2ServoPower				:=	FALSE;*)
					//END_IF	
					iCountAborting	:=	iCountAborting	+	1;						
				20: //Stop Done
					IF 
						(mcHeightStop.Done 		OR NOT bHeightServoPower	) AND 
						(mcScrewer1Stop.Done 	OR NOT bScrewer1ServoPower	OR NOT bEnable1) AND 
						(mcScrewer2Stop.Done 	OR NOT bScrewer2ServoPower	OR NOT bEnable2)
						 THEN
							bHeightServoPower		:=	FALSE;
							bScrewer1ServoPower		:=	FALSE;
							bScrewer2ServoPower		:=	FALSE;		
							iAbortingCASE			:=	iAbortingCASE	+	10;			
					END_IF	
					
				30: //Wyjście
					ResetCommands(); 
					eState							:=	E_Station.eAborted; 
					eRunningState					:=	E_GripperScrewer.eReady;
			END_CASE
			
	/////////////////////////////			
		E_Station.eError:                 	 	// Stan błędu 	
			
			mcHeightMoveAbsolute.Execute 	:= FALSE;

			IF bReset THEN
				eState 						:= E_Station.eResetting;
				iTestResetting					:= iTestResetting	+	1;
			ELSIF tonError.Q THEN
				ResetCommands();
			END_IF
			
	/////////////////////////////
		E_Station.eResetting:					// Stan resetowania bledu (po Errorze)

			//Procedura obsługi resetu w zależności od błędu
//			CASE udiErrorID OF
//			CASE udiErrorID-iStationIndex OF
			
				//Error 2 - BŁĄD SERWA PODNOSZENIA ZAKRĘCARKI
				//Error 5 - BŁĄD NASTAW MAX			
// 				295:	
// 					fbHeightHardReset						(Execute:=NOT mcHeightMoveAbsolute.Execute,	Axis:=HeightAxisRef);
// 					mcHeightSoftReset						(Execute:=TRUE,								Axis:=HeightAxisRef);																		
// 					IF NOT fbHeightHardReset.Busy AND NOT mcHeightSoftReset.Busy AND mcHeightPower.Status AND NOT HeightAxisRef.Status.Error THEN
// 						fbHeightHardReset					(Execute:=FALSE,							Axis:=HeightAxisRef);
// 						mcHeightSoftReset					(Execute:=FALSE,							Axis:=HeightAxisRef);
// 						mcHeightMoveAbsolute.Velocity		:=	lrHeightSpeed;
// 						mcHeightMoveAbsolute.Position		:=	lrHeightReadyPosition; 
// 						mcHeightMoveAbsolute.Execute		:=	TRUE;
// 						IF mcHeightMoveAbsolute.Done THEN
// 							mcHeightMoveAbsolute.Execute	:=	FALSE;
// 							mcHeightPower.Override			:=	100;
// 							mcScrewing1Power.Override		:=	100;
// 							mcScrewing2Power.Override		:=	100;
// 							bError							:=	FALSE;
// 							udiHeightServoErrorNr			:=	0;
// 							sErrorDescription				:=	'';	
// 							udiErrorID						:=	0;	
// 						END_IF
// 					ELSIF NOT fbHeightHardReset.Busy AND NOT mcHeightSoftReset.Busy AND NOT mcHeightPower.Status AND NOT HeightAxisRef.Status.Error  THEN
// 						fbHeightHardReset					(Execute:=FALSE,							Axis:=HeightAxisRef);
// 						mcHeightSoftReset					(Execute:=FALSE,							Axis:=HeightAxisRef);
// 						mcHeightPower.Override				:=	100;
// 						mcScrewing1Power.Override			:=	100;
// 						mcScrewing2Power.Override			:=	100;
// 						bError 								:=	FALSE;
// 						udiHeightServoErrorNr				:=	0;
// 						sErrorDescription					:=	'';	
// 						udiErrorID							:=	0;		  	
// 					END_IF
					
				//Error 3 - BŁĄD SERWA ZAKRĘCAJĄCEGO 1
				//Error 4 - BŁĄD SERWA ZAKRĘCAJĄCEGO 2
		IF arfbAlarm[0].bActive OR arfbAlarm[1].bActive OR arfbAlarm[2].bActive OR arfbAlarm[3].bActive OR arfbAlarm[4].bActive THEN				
		//		291, 292, 293,294:	
 					CASE iErrorResseting3 OF
					0:
						IF NOT mcHeightPower.Status THEN
							bHeightServoPower := FALSE;
						END_IF				
						(*IF NOT mcScrewing1Power.Status THEN
							bScrewer1ServoPower := FALSE;
						END_IF
						IF NOT mcScrewing2Power.Status THEN
							bScrewer2ServoPower := FALSE;
						END_IF*)
						IF NOT mcScrewing1Power.Status OR NOT mcScrewing2Power.Status THEN
							bScrewer1ServoPower := FALSE;
							bScrewer2ServoPower := FALSE;
						END_IF
						(*fbScrewer1HardReset					(Execute:=bEnable1,	Axis:=Screwing1AxisRef);
						mcScrewer1SoftReset					(Execute:=bEnable1,	Axis:=Screwing1AxisRef);
						fbScrewer2HardReset					(Execute:=bEnable2,	Axis:=Screwing2AxisRef);
						mcScrewer2SoftReset					(Execute:=bEnable2,	Axis:=Screwing2AxisRef);		*)
						//Zmiana LU207
						fbScrewer1HardReset					(Execute:=TRUE,	Axis:=Screwing1AxisRef);
						mcScrewer1SoftReset					(Execute:=TRUE,	Axis:=Screwing1AxisRef);
						fbScrewer2HardReset					(Execute:=TRUE,	Axis:=Screwing2AxisRef);
						mcScrewer2SoftReset					(Execute:=TRUE,	Axis:=Screwing2AxisRef);		
						
						
						mcHeightGearOut.Execute				:= TRUE;	
						fbHeightHardReset					(Execute:=TRUE,		Axis:=HeightAxisRef); 
						mcHeightSoftReset					(Execute:=TRUE,		Axis:=HeightAxisRef);
				
						iErrorResseting3					:=	10;
						iTestError3:=iTestError3+1;
						
					10:	 // na próbe
						IF bEnable1 THEN
							bScrewer1ServoPower := TRUE;
							bHeightServoPower 	:= TRUE;// test xts
						END_IF
						
						IF bEnable2 THEN
							bScrewer2ServoPower := TRUE;
														bHeightServoPower 	:= TRUE;// test xts

						END_IF		
						iErrorResseting3					:=	20;
					20:
						IF 
						( NOT fbScrewer1HardReset.Busy AND NOT mcScrewer1SoftReset.Busy AND (mcScrewing1Power.Status OR NOT bEnable1) AND NOT Screwing1AxisRef.Status.Error ) AND
						( NOT fbScrewer2HardReset.Busy AND NOT mcScrewer2SoftReset.Busy AND (mcScrewing2Power.Status OR NOT bEnable2) AND NOT Screwing2AxisRef.Status.Error ) AND
						( NOT fbHeightHardReset.Busy AND NOT mcHeightSoftReset.Busy AND mcHeightPower.Status  AND NOT HeightAxisRef.Status.Error )
						
						THEN
							fbScrewer1HardReset					(Execute:=FALSE,	Axis:=Screwing1AxisRef);
							mcScrewer1SoftReset					(Execute:=FALSE,	Axis:=Screwing1AxisRef);
							fbScrewer2HardReset					(Execute:=FALSE,	Axis:=Screwing2AxisRef);
							mcScrewer2SoftReset					(Execute:=FALSE,	Axis:=Screwing2AxisRef);
							mcHeightGearOut.Execute				:= FALSE;
							fbHeightHardReset					(Execute:=FALSE,	Axis:=HeightAxisRef); 
							mcHeightSoftReset					(Execute:=FALSE,	Axis:=HeightAxisRef);	
							mcHeightMoveAbsolute.Velocity		:=	lrHeightSpeed;						
							mcHeightMoveAbsolute.Position		:=	lrHeightReadyPosition; 	
							mcHeightMoveAbsolute.Execute		:=	TRUE;


							IF mcHeightMoveAbsolute.Done THEN
								mcHeightMoveAbsolute.Execute	:=	FALSE;
								mcHeightPower.Override			:=	100;
								mcScrewing1Power.Override		:=	100;
								bError							:=	FALSE;
								iErrorResseting3				:=	0;
								udiScrewing1ServoErrorNr		:=	0;
								sErrorDescription				:=	'';	
								udiErrorID						:=	0;
							END_IF 	
						ELSIF 
						( NOT fbScrewer1HardReset.Busy	AND NOT mcScrewer1SoftReset.Busy AND NOT mcScrewing1Power.Status AND NOT bScrewer1ServoPower AND NOT Screwing1AxisRef.Status.Error ) AND
						( NOT fbScrewer2HardReset.Busy	AND NOT mcScrewer2SoftReset.Busy AND NOT mcScrewing2Power.Status AND NOT bScrewer2ServoPower AND NOT Screwing2AxisRef.Status.Error ) AND
						( NOT fbHeightHardReset.Busy	AND NOT mcHeightSoftReset.Busy 									AND NOT mcHeightPower.Status  AND NOT HeightAxisRef.Status.Error )
		
					THEN
							fbScrewer1HardReset					(Execute:=FALSE,	Axis:=Screwing1AxisRef);
							mcScrewer1SoftReset					(Execute:=FALSE,	Axis:=Screwing1AxisRef);
							fbScrewer2HardReset					(Execute:=FALSE,	Axis:=Screwing2AxisRef);
							mcScrewer2SoftReset					(Execute:=FALSE,	Axis:=Screwing2AxisRef);
							fbHeightHardReset					(Execute:=FALSE,	Axis:=HeightAxisRef); 
							mcHeightSoftReset					(Execute:=FALSE,	Axis:=HeightAxisRef);						
							mcHeightPower.Override				:=	100;
							mcScrewing1Power.Override			:=	100;
							bError								:=	FALSE;
							iErrorResseting3					:=	0;	
							udiScrewing1ServoErrorNr			:=	0;
							sErrorDescription					:=	'';
							udiErrorID							:=	0;
						END_IF	
					END_CASE
			END_IF	
// 				//Error 6 - BŁAD POZYCJI MINIMALNEJ PODNOŚNIKA 
// 				296:
// 					mcHeightStop.Execute						:=	FALSE;
// 					sErrorDescription							:=	'';	
// 					udiErrorID									:=	0;					
// 					eState										:=	E_Station.eReady;
// 				ELSE
// 					bError					:=	FALSE;	
// 				END_CASE	
			
			IF NOT bError THEN
				udiErrorID 						:=	0;
   				sErrorDescription 				:=	'';                       			
				eState 							:=	E_Station.ePreparingToReady;
			ELSIF tonResetting.Q THEN            	
				eState 							:=	E_Station.eError;
			END_IF
        
	/////////////////////////////
		E_Station.eManualMovement:     			// Stan ruchów manualnych  
       
			ManualMovements();
			//Wyjście z trybu serwisowego
			IF NOT bManualMovement THEN
					bManualGripper1				:=	FALSE;
					bManualGripper2				:=	FALSE;		
					bGripper1Actuator			:=	FALSE;
					bGripper2Actuator			:=	FALSE;	
			
					mcHeightPower.Override		:=	100;
					mcScrewing1Power.Override	:=	100;
					mcScrewing2Power.Override	:=	100;
	
					IF HeightAxisRef.NcToPlc.ActPos	<	lrHeightReadyPosition-1 THEN
						bHomingDone							:=	FALSE;
						mcHeightMoveAbsolute.Execute		:=	TRUE;
						mcHeightMoveAbsolute.Position		:=	lrHeightReadyPosition;
						mcHeightMoveAbsolute.Velocity		:=	100;
						IF mcHeightMoveAbsolute.Done THEN
							mcHeightMoveAbsolute.Execute	:=	FALSE;
							eState							:=	E_Station.eReady;
						END_IF	
					ELSE
							eState							:=	E_Station.eReady;
					END_IF	
			END_IF

	/////////////////////////////
		E_Station.eHoming:						// Stan bazowania 

			Homing();
			IF NOT bHoming AND NOT bHeightSet THEN
			  	eState							:=	E_Station.ePreparingToReady;
			   	mcHeightManualMove.JogForward	:=	FALSE;
				mcHeightManualMove.JogBackwards	:=	FALSE;
			END_IF		
			
	/////////////////////////////
		E_Station.eHomingDone:                  // Stan wykonania bazowania 
		
			bHeighSetNotDone 					:=	FALSE;
			mcHeightManualMove.JogForward		:=	FALSE;
			mcHeightManualMove.JogBackwards		:=	FALSE;
			bHomingDone							:=	TRUE;
			IF NOT bHoming AND NOT bHeightSet THEN
			   	eState							:=	E_Station.eReady;
			END_IF
			
	/////////////////////////////
		E_Station.ePreparingToReady:            // Stan przygotowywania do gotowosci (zawsze przed Ready)  
			
			rScrewing1ProportionalGain	:= 10;
			rScrewing2ProportionalGain	:= 10;		
		
			CASE iPreparingToReadyCase OF
		
			0:
			
				bGripper1Actuator				:=	FALSE;
				bGripper2Actuator				:=	FALSE;
				IF tonDelayServoOn.Q THEN
					bHeightServoPower			:=	TRUE;	// Przy pierwszym uruchomieniu Ustawienia Fabryczne robimy na wartość maksymalną
					bScrewer1ServoPower			:=	bEnable1;
					bScrewer2ServoPower			:=	bEnable2;
					iPreparingToReadyCase		:=	iPreparingToReadyCase	+	10;	
				END_IF	
				
			10:	//Dalej jak serwa się włączyły

				IF mcHeightPower.Status AND (mcScrewing1Power.Status OR NOT bEnable1) AND (mcScrewing2Power.Status OR NOT bEnable2) THEN 
					iPreparingToReadyCase				:= 12;
				END_IF
			
			12: //Rozgearowanie
	
				IF mcHeightGearInMultiMaster.InGear THEN
					mcHeightGearInMultiMaster.Enable 	:=	FALSE;
					mcHeightGearOut.Execute 			:=	TRUE;
				ELSIF mcHeightGearInMultiMaster.Enable AND mcHeightGearOut.Done THEN 
					mcHeightGearOut.Execute 			:=	FALSE;
				ELSE
					bHeighSetNotDone					:=	FALSE;
					mcHeightMoveAbsolute.Execute		:=	FALSE;
					iPreparingToReadyCase				:=	14;
				END_IF	
	
			14:
				iPreparingToReadyCase					:= 20;
				
			20: //Obrót 1
				IF 		M_PrepareToReady(	AxisRef			:=  Screwing1AxisRef,	(*Obrót*) 		
											iGripperArms	:=	2					)			OR NOT bEnable1
				THEN
					iPreparingToReadyCase					:= iPreparingToReadyCase	+	10;	
				END_IF
			
			30: //Obrót 2
				IF 		M_PrepareToReady(	AxisRef			:=  Screwing2AxisRef,	(*Obrót*) 		
											iGripperArms	:=	2					)			OR NOT bEnable2
				THEN
					iPreparingToReadyCase					:= iPreparingToReadyCase	+	10;	
				END_IF
			
			40:	//Koniec
				eState							:=	E_Station.eReady;
				eRunningState					:=	E_GripperScrewer.eReady;
				iPreparingToReadyCase			:= 0;
			
			END_CASE
				

         	IF bIgnoreError THEN
				eState										:=	E_Station.eReady;
				eRunningState								:=	E_GripperScrewer.eReady;
			END_IF
			
	/////////////////////////////
		E_Station.ePreparingToDisable:          // Stan przygotowywania do nieaktywnosci (po wyłączeniu Enable) 
  
			bHeightServoPower		:=	TRUE;			// Przy pierwszym uruchomieniu Ustawienia Fabryczne robimy na wartość maksymalną
			bScrewer1ServoPower		:=	TRUE;
			bScrewer2ServoPower		:=	TRUE;
			bGripper1Actuator		:=	FALSE;
			bGripper2Actuator		:=	FALSE;	
		
			IF bPreparingToDisable THEN
				IF mcHeightPower.Status AND (mcScrewing1Power.Status OR NOT bEnable1) AND (mcScrewing2Power.Status OR NOT bEnable2) THEN
					mcHeightPower.Override				:=	10;
					mcHeightMoveAbsolute.Velocity		:=	100;
					mcHeightMoveAbsolute.Position		:=	lrMaxHeightPosition;
					mcHeightMoveAbsolute.Execute		:=	TRUE;
					IF mcHeightMoveAbsolute.Done THEN
						mcHeightMoveAbsolute.Execute	:=	FALSE;
						mcScrewer1SoftReset				(Axis:=Screwing1AxisRef, Execute:=FALSE); //LU205
						mcScrewer2SoftReset				(Axis:=Screwing2AxisRef, Execute:=FALSE); //LU205
						bScrewer1ServoPower				:=	FALSE;//LU205
						bScrewer2ServoPower				:=	FALSE;//LU205
						bHeightServoPower				:=	FALSE;//LU205
						eState							:=	E_Station.eDisabled;
						eRunningState					:=	E_GripperScrewer.eReady;
					END_IF	
				END_IF
			ELSE
				mcScrewer1Stop.Execute	:=	bEnable1;
				mcScrewer2Stop.Execute	:=	bEnable2;				
				IF (mcScrewer1Stop.Done OR mcScrewer1Stop.CommandAborted OR NOT bEnable1) AND (mcScrewer2Stop.Done OR mcScrewer2Stop.CommandAborted OR NOT bEnable2) THEN							
					IF HeightAxisRef.NcToPlc.CoupleState	<	3 THEN
						mcHeightGearOut.Execute						:=	FALSE;
						mcHeightGearInMultiMaster.Enable			:=	FALSE;			
						mcHeightMoveAbsolute.Execute				:=	FALSE;
						mcHeightStop.Execute						:=	FALSE;
						mcScrewer1Stop.Execute 						:=	FALSE;
						mcScrewer2Stop.Execute 						:=	FALSE;		
						bPreparingToDisable							:=	TRUE;				
					ELSIF HeightAxisRef.NcToPlc.CoupleState	=	3 THEN
						mcHeightGearInMultiMaster.Enable			:=	FALSE;
						mcHeightGearOut.Execute						:=	TRUE;
					END_IF
				END_IF
			END_IF
			
         	IF bIgnoreError THEN
				eState:=E_Station.eDisabled;
				eRunningState:=E_GripperScrewer.eReady;
			END_IF
			
	/////////////////////////////
		E_Station.eReady:						// Stan gotowosci 
			
			(*Skasowanie wszystkich komend*)
			IF rtResetCommands.Q THEN	ResetCommands();	END_IF
		
			IF (bRun1 OR bRun2) AND NOT bCycleDone1 AND NOT bCycleNotDone1 AND NOT bCycleDone2 AND NOT bCycleNotDone2 THEN
				eState 				:= E_Station.eStarting; 
			END_IF
			IF bHoming OR bHeightSet THEN
				eState 				:= E_Station.eHoming; 
			END_IF
			IF bManualMovement THEN
				//Jeśli przejście w tryb ruchów manualnych przepisz wszystkie stany siłowników sterowanych przez moduł
				//aby zapobiec ewentualnym kolizjom po wejściu w tryb serwisowy
				bManualGripper1				:=	bGripper1Actuator;
				bManualGripper2				:=	bGripper2Actuator;
				mcScrewer1Stop.Execute		:=	FALSE;
				mcScrewer2Stop.Execute		:=	FALSE;				
				eState 						:=	E_Station.eManualMovement; 
			END_IF
			IF NOT bRun1 AND NOT bRun2 THEN
				bCycleDone1 				:= FALSE;
				bCycleNotDone1 				:= FALSE;	
				bCycleDone2					:= FALSE;
				bCycleNotDone2 				:= FALSE;	
				bWarning1					:= FALSE;	
				bWarning2					:= FALSE;	
			END_IF
			
			
	/////////////////////////////
		E_Station.eStopping:					// Stan zatrzymywania 
			
			Running();
			bGripper1Actuator 					:=	FALSE;
			bGripper2Actuator 					:=	FALSE;		
	
			IF NOT  bHeightGearingWithScrewer THEN 	(* Wersja bez gearowania*)
				CASE iStoppingCase OF
					0:
						mcHeightStop.Execute				:=	TRUE;
						mcHeightMoveAbsolute.Velocity		:=	lrHeightSpeed;	
						mcHeightMoveAbsolute.Position		:=	lrHeightReadyPosition;	
									
						mcScrewer1Stop.Execute				:=	bEnable1;
						mcScrewer2Stop.Execute				:=	bEnable2;
						mcScrewer1MoveRelative.Execute		:=	FALSE;
						mcScrewer1MoveVelocity.Execute		:=	FALSE;
						mcScrewer1MoveVelocity2.Execute		:=	FALSE;		
						mcScrewer1MoveVelocity3.Execute		:=	FALSE;					
						mcScrewer2MoveRelative.Execute		:=	FALSE;
						mcScrewer2MoveVelocity.Execute		:=	FALSE;
						mcScrewer2MoveVelocity2.Execute		:=	FALSE;						
						mcScrewer2MoveVelocity3.Execute		:=	FALSE;									
						uiScrewing1TorqueControl			:=	0; // bylo 6000	
						mcScrewer1SoftReset					(Axis:=Screwing1AxisRef, Execute:= bEnable1);
						uiScrewing2TorqueControl			:=	0; // bylo 6000	
						mcScrewer2SoftReset					(Axis:=Screwing2AxisRef, Execute:= bEnable2);
						
						IF 	mcHeightStop.Done AND	(mcScrewer1Stop.Done OR mcScrewer1Stop.CommandAborted OR NOT bEnable1) AND
													(mcScrewer2Stop.Done OR mcScrewer2Stop.CommandAborted OR NOT bEnable2)
						 THEN	
							iStoppingCase := iStoppingCase + 10;
						END_IF
						
					10:	
						mcHeightMoveAbsolute.Execute		:=	tonGripper1ReliseDelay.Q AND tonGripper2ReliseDelay.Q;
						IF 	mcHeightMoveAbsolute.Done  THEN
							mcHeightMoveAbsolute.Execute	:=	FALSE;
							iStoppingCase 						:=	iStoppingCase + 10;
						END_IF
					20:
						iStoppingCase 							:=	0;
						eState 								:=	E_Station.eReady;

				END_CASE
			ELSE									(* Wersja z gearowaniem*)
				CASE iStoppingCase OF
					0: //STOP OSI
						IF mcHeightGearInMultiMaster.InGear THEN
							mcScrewer1Stop.Execute				:=	bEnable1;
							mcScrewer1MoveRelative.Execute		:=	FALSE;
							mcScrewer1MoveVelocity.Execute		:=	FALSE;
							mcScrewer1MoveVelocity2.Execute		:=	FALSE;
							mcScrewer1MoveVelocity3.Execute		:=	FALSE;							
							uiScrewing1TorqueControl			:=	0; 					
							
							mcScrewer2Stop.Execute				:=	bEnable2;
							mcScrewer2MoveRelative.Execute		:=	FALSE;
							mcScrewer2MoveVelocity.Execute		:=	FALSE;
							mcScrewer2MoveVelocity2.Execute		:=	FALSE;
							mcScrewer2MoveVelocity3.Execute		:=	FALSE;							
							uiScrewing2TorqueControl			:=	0; 								
					
							IF (mcScrewer1Stop.Done OR mcScrewer1Stop.CommandAborted OR NOT bEnable1) AND (mcScrewer2Stop.Done OR mcScrewer2Stop.CommandAborted OR NOT bEnable2) THEN
								mcScrewer1Stop.Execute			:=	FALSE;	
								mcScrewer2Stop.Execute			:=	FALSE;									
								iStoppingCase						:=	iStoppingCase + 10;
							END_IF
						ELSE
							mcScrewer1Stop.Execute				:=	bEnable1;
							mcScrewer2Stop.Execute				:=	bEnable2;							
							mcHeightStop.Execute				:=	TRUE;
							IF 	mcHeightStop.Done AND (mcScrewer1Stop.Done OR mcScrewer1Stop.CommandAborted OR NOT bEnable1) AND (mcScrewer2Stop.Done OR mcScrewer2Stop.CommandAborted OR NOT bEnable2)THEN
								mcHeightStop.Execute			:=	FALSE;
								mcScrewer1Stop.Execute			:=	FALSE;
								mcScrewer2Stop.Execute			:=	FALSE;
								iStoppingCase 						:=	20;
							END_IF	
						END_IF	
							
					10: //GEAR OUT
						mcHeightGearInMultiMaster.Enable		:=	FALSE;
						mcHeightGearOut.Execute					:=	TRUE;
						IF mcHeightGearOut.Done THEN        	
							mcHeightGearOut.Execute				:=	FALSE;
							iStoppingCase 							:= iStoppingCase + 10;
						END_IF
						
					20: //Podjazd do góry i reset laga
					
						uiScrewing1TorqueControl			:=	0; 
						uiScrewing2TorqueControl			:=	0; 
				
						mcHeightMoveAbsolute.Velocity		:=	lrHeightSpeed;	
						mcHeightMoveAbsolute.Position		:=	lrHeightReadyPosition;	
						mcHeightMoveAbsolute.Execute		:=	(tonGripper1ReliseDelay.Q AND tonGripper1ReliseDelay.Q); 
						
						//Reset laga			
						mcScrewer1SoftReset.Execute			:= bEnable1;
						mcScrewer2SoftReset.Execute			:= bEnable2;	
									
						//Sprawdzanie czy lag się zresetował
						IF	(mcScrewer1SoftReset.Done OR NOT bEnable1) AND
							(mcScrewer2SoftReset.Done OR NOT bEnable2) //AND
							 //Screwing1AxisRef.NcToPlc.PosDiff < 5 AND Screwing2AxisRef.NcToPlc.PosDiff < 5 AND
							AND	mcHeightMoveAbsolute.Done  THEN
								mcScrewer1SoftReset.Execute		:= FALSE;
								mcScrewer2SoftReset.Execute		:= FALSE;
								mcHeightMoveAbsolute.Execute	:=	FALSE;
								iStoppingCase					:= iStoppingCase	+	10;					
						END_IF					
				
					30: //Obrót 1
						IF 		M_PrepareToReady(	AxisRef			:=  Screwing1AxisRef,	(*Obrót*) 		
													iGripperArms	:=	2					)			OR NOT bEnable1
						THEN
							iStoppingCase							:= iStoppingCase	+	10;	
						END_IF
					
					40: //Obrót 2
						IF 		M_PrepareToReady(	AxisRef			:=  Screwing2AxisRef,	(*Obrót*) 		
													iGripperArms	:=	2					)			OR NOT bEnable2
						THEN
							iStoppingCase							:= iStoppingCase	+	10;	
						END_IF
					
					50:	//Koniec
						eState 										:=	E_Station.eReady;
						iStoppingCase								:= 0;
										
				END_CASE
			END_IF
				
				
	/////////////////////////////
		E_Station.eStarting:                  	// Stan uruchamiania (po Ready)
					
			eState		:= E_Station.eRunning; 
			
	/////////////////////////////
		E_Station.eRunning:               		// Stan wykonywania cyklu (po Startingu), w tym stanie osobny
 
			Running();
			IF NOT bRun1 AND NOT bRun2 THEN					(*Przerywanie cyklu*)
				eState 				 := E_Station.eStopping;	
			END_IF
			IF (bCycleDone1 OR bCycleNotDone1) AND (bCycleDone2 OR bCycleNotDone2)  THEN (*Cykl zakończony*)
				eState 				 := E_Station.eReady;
			END_IF	
			
			
	/////////////////////////////		
	END_CASE
END_ACTION

ACTION ErrorHandling:
// Alarm_0460	460	Error	Błąd napędu podnoszenia. Błąd NC: {0}
// Alarm_0461	461	Error	Błąd napędu zakręcającego 1. Błąd NC: {0}
// Alarm_0462	462	Error	Błąd napędu zakręcającego 2. Błąd NC: {0}
// Alarm_0463	463	Error	Wartość zadana wysokości jest większa od maksymalnej - zmień ustawienia w recepturze {0}
// Alarm_0464	464	Error	Wartość zadana wysokości jest mniejsza od minimalnej - zmień ustawienia w recepturze {0}
// Alarm_0465	465	Error	Zbyt wysoka temperatura napędu zakręcającego 1 > 130C - zmniejsz moment zakręcania
// Alarm_0466	466	Error	Zbyt wysoka temperatura napędu zakręcającego 2 > 130C - zmniejsz moment zakręcania

IF bAlarmInit THEN
    bAlarmInit := FALSE; 
	fbSourceInfo.Clear();
	fbSourceInfo.sName:=wsLiteral_TO_UTF8(sStationName);//'Machine';
	fbSourceInfo.nId:=iStationIndex;//2700;
	// Alarm_0460	460	Error	Błąd napędu podnoszenia. Błąd NC: {0}
    arfbAlarm[0].CreateEx(stEventEntry := TC_EVENTS.AlarmClass.Alarm_0460, bWithConfirmation:= FALSE,  ipSourceInfo:= fbSourceInfo); 
	// Alarm_0461	461	Error	Błąd napędu zakręcającego 1. Błąd NC: {0}
	arfbAlarm[1].CreateEx(stEventEntry := TC_EVENTS.AlarmClass.Alarm_0461, bWithConfirmation:= FALSE,  ipSourceInfo:= fbSourceInfo);
	// Alarm_0462	462	Error	Błąd napędu zakręcającego 2. Błąd NC: {0}
	arfbAlarm[2].CreateEx(stEventEntry := TC_EVENTS.AlarmClass.Alarm_0462, bWithConfirmation:= FALSE,  ipSourceInfo:= fbSourceInfo);
	// Alarm_0463	463	Error	Wartość zadana wysokości jest większa od maksymalnej - zmień ustawienia w recepturze {0}
	arfbAlarm[3].CreateEx(stEventEntry := TC_EVENTS.AlarmClass.Alarm_0463, bWithConfirmation:= FALSE,  ipSourceInfo:= fbSourceInfo);
	// Alarm_0464	464	Error	Wartość zadana wysokości jest mniejsza od minimalnej - zmień ustawienia w recepturze {0}
	arfbAlarm[4].CreateEx(stEventEntry := TC_EVENTS.AlarmClass.Alarm_0464, bWithConfirmation:= FALSE,  ipSourceInfo:= fbSourceInfo);
	// Alarm_0465	465	Error	Zbyt wysoka temperatura napędu zakręcającego 1 > 130C - zmniejsz moment zakręcania
	arfbAlarm[5].CreateEx(stEventEntry := TC_EVENTS.AlarmClass.Alarm_0465, bWithConfirmation:= FALSE,  ipSourceInfo:= fbSourceInfo);
	// Alarm_0466	466	Error	Zbyt wysoka temperatura napędu zakręcającego 2 > 130C - zmniejsz moment zakręcania
	arfbAlarm[6].CreateEx(stEventEntry := TC_EVENTS.AlarmClass.Alarm_0466, bWithConfirmation:= FALSE,  ipSourceInfo:= fbSourceInfo);
	
END_IF



//CZYTANIE STATUSÓW

HeightAxisRef.ReadStatus();
Screwing1AxisRef.ReadStatus();
Screwing2AxisRef.ReadStatus();

//**********************LISTA BŁĘDÓW******************************
bStateError	:= (eState=E_Station.eError) OR (eState=E_Station.eResetting) OR NOT bEstop OR bIgnoreError;

//PreparingToDisable i StateError ze względu na wciśnięcie EStopa podczas wyłączania i pojawienie się blędu
IF bEnable1 OR bEnable2 OR (eState=E_Station.ePreparingToDisable OR bStateError) THEN
	
	//Warning 1 - ZA DŁUGIE ZAKRĘCANIE ZAKRĘCARKĄ 1
	tonTooLongScrewing1			(IN:=eRunningState=E_GripperScrewer.eScrewing 		AND bRun1 AND NOT bScrewed1,											PT:=tTooLongScrewing1);//bylo 2
	tonTooLongFinding1			(IN:=eRunningState=E_GripperScrewer.eFindingScrew 	AND bRun1,																PT:=T#5S);//bylo 2
	tonPosDiff1Error			(IN:=ABS(Screwing1AxisRef.NcToPlc.ActPos-lrStartPosition1)>=6080 AND eRunningState=E_GripperScrewer.eScrewing AND bRun1,	PT:=T#1MS);//bylo 1ms
//	tonPosTooLowWhenScrewing1	(IN:=eRunningState=E_GripperScrewer.eScrewing 		 AND ABS(HeightAxisRef.NcToPlc.ActPos)<lrMinHeightPosition+2);
	tonPosTooLowWhenScrewing1.PT;
	IF iTool <>4 THEN // Różna od zasysającej
		IF iTool = 2 THEN //Glowica ksztaltowa
			(*tonPosTooLowWhenScrewing1	(IN:=bRun1 AND eRunningState=E_GripperScrewer.eScrewing 		 AND 
									(
										ABS(ABS(lrStartPosition1)-ABS(Screwing1AxisRef.NcToPlc.SetPos))> (lrPackageTurnoversToFullScrewed*360.0*5)  AND 
										NOT tonTightScrewing1Timer.Q
									));	*)
			tonPosTooLowWhenScrewing1	(IN:=bRun1 AND eRunningState=E_GripperScrewer.eScrewing 		 AND 
									(
										ABS(HeightAxisRef.NcToPlc.ActPos)<lrHeightEndScrewingPosition-30 OR 
										ABS(HeightAxisRef.NcToPlc.ActPos-iToolHeight)<lrMinHeightPosition+2)
									);						
									
		ELSE
			tonPosTooLowWhenScrewing1	(IN:=bRun1 AND eRunningState=E_GripperScrewer.eScrewing 		 AND 
										(
										ABS(HeightAxisRef.NcToPlc.ActPos)<lrHeightEndScrewingPosition-(*20*) 25 OR  //bylo 50
										//ABS(HeightAxisRef.NcToPlc.ActPos)<lrMinHeightPosition+2)
										ABS(HeightAxisRef.NcToPlc.ActPos-iToolHeight)<lrMinHeightPosition-5)										
										);
		END_IF
	ELSE
		tonPosTooLowWhenScrewing1	(IN:=bRun1 AND eRunningState=E_GripperScrewer.eScrewing 		 AND 
								(
								//ABS(HeightAxisRef.NcToPlc.ActPos)<lrHeightEndScrewingPosition-20 OR 
								ABS(HeightAxisRef.NcToPlc.ActPos-iToolHeight)<lrMinHeightPosition-50)
								);		
	END_IF
	
	IF (tonTooLongScrewing1.Q OR tonTooLongFinding1.Q OR tonPosDiff1Error.Q OR tonPosTooLowWhenScrewing1.Q) AND NOT bStateError THEN
		//bGripper1Actuator				:=	FALSE;
		mcScrewer1MoveVelocity.Execute	:=	FALSE;
		(*Kasownie momentu po zakręceniu, zeby nie było samoistnego wrócenia do pozycji*)
		uiScrewing1TorqueControl		:=	0; 
		//mcScrewer1SoftReset				(Axis:=Screwing1AxisRef, Execute:= TRUE);
		bWarning1						:=	TRUE;			
		udiWarningID					:= 1;
		IF tonTooLongScrewing1.Q THEN
			sWarningDescription				:=	'Zakręcarka 1 - przekroczenie czasu zakręcania - zmień ust.';
			bWarning1A						:= TRUE;
		END_IF
		IF tonTooLongFinding1.Q THEN
			sWarningDescription				:=	'Zakręcarka 1 - przekroczenie czasu szukania gwintu - zmień ust.';
			bWarning1B						:= TRUE;
		END_IF
		IF tonPosDiff1Error.Q THEN
			sWarningDescription				:=	'Zakręcarka 1 - przekroczenie laga - zmień ust.';
			bWarning1C						:= TRUE;
		END_IF
		IF tonPosTooLowWhenScrewing1.Q THEN
			sWarningDescription				:=	'Zakręcarka 1 - zbyt niska pozycja przy zakrecaniu - zmień ust.';
			bWarning1D						:= TRUE;
		END_IF	
	END_IF
	
	//Warning 1E - Nie znaleziono gwintu podczas jego szukania z czujnikiem
	(*Generowanie ostrzeżenia*)
	IF bOptionFindScrewWithHeightSensor AND mcScrewer1MoveRelative.Done AND (iFindingScrewCASE	=	40 OR iFindingScrewCASE	=	50) AND NOT bStateError THEN
		bWarning1E						:= TRUE;
		udiWarningID					:=	1;
		sWarningDescription				:=	'Zakręcarka 1 - nie znaleziono początku gwintu';
	END_IF
	
	
	//Warning 2 - ZA DŁUGIE ZAKRĘCANIE ZAKRĘCARKĄ 2
	tonTooLongScrewing2			(IN:=eRunningState=E_GripperScrewer.eScrewing 		AND bRun2 AND NOT bScrewed2,											PT:=tTooLongScrewing2);//bylo 2
	tonTooLongFinding2			(IN:=eRunningState=E_GripperScrewer.eFindingScrew 	AND bRun2,																PT:=T#5S);//bylo 2
	tonPosDiff2Error			(IN:=ABS(Screwing2AxisRef.NcToPlc.ActPos-lrStartPosition2)>=6080 AND eRunningState=E_GripperScrewer.eScrewing AND bRun2,	PT:=T#1MS);//bylo 1ms
	tonPosTooLowWhenScrewing2.PT;
	IF iTool <>5 THEN // Różna od zasysającej
		IF iTool = 2 THEN
			(*tonPosTooLowWhenScrewing2	(IN:=bRun2 AND eRunningState=E_GripperScrewer.eScrewing 		 AND 
									(
										ABS(ABS(lrStartPosition2)-ABS(Screwing2AxisRef.NcToPlc.SetPos))> (lrPackageTurnoversToFullScrewed*360.0*1.5)  AND
										NOT tonTightScrewing2Timer.Q
									));	*)
			tonPosTooLowWhenScrewing2	(IN:=bRun2 AND eRunningState=E_GripperScrewer.eScrewing 		 AND 
									(
									ABS(HeightAxisRef.NcToPlc.ActPos)<lrHeightEndScrewingPosition-30 OR 
									ABS(HeightAxisRef.NcToPlc.ActPos)<lrMinHeightPosition+2)
									);							
									
		ELSE
			tonPosTooLowWhenScrewing2	(IN:=bRun2 AND eRunningState=E_GripperScrewer.eScrewing 		 AND 
									(
									ABS(HeightAxisRef.NcToPlc.ActPos)<lrHeightEndScrewingPosition-(*20*) 50 OR 
//									ABS(HeightAxisRef.NcToPlc.ActPos)<lrMinHeightPosition+2)
									ABS(HeightAxisRef.NcToPlc.ActPos)<lrMinHeightPosition-5)									
									);
		END_IF
	ELSE
		tonPosTooLowWhenScrewing2	(IN:=bRun2 AND eRunningState=E_GripperScrewer.eScrewing 		 AND 
									(
									//ABS(HeightAxisRef.NcToPlc.ActPos)<lrHeightEndScrewingPosition-20 OR 
									ABS(HeightAxisRef.NcToPlc.ActPos)<lrMinHeightPosition-50)
									);	
	END_IF
	
	IF (tonTooLongScrewing2.Q OR tonTooLongFinding2.Q OR tonPosDiff2Error.Q OR tonPosTooLowWhenScrewing2.Q) AND NOT bStateError THEN
		bGripper2Actuator				:=	FALSE;
		mcScrewer2MoveVelocity.Execute	:=	FALSE;
		(*Kasownie momentu po zakręceniu, zeby nie było samoistnego wrócenia do pozycji*)
		uiScrewing2TorqueControl		:=	0; 
		//mcScrewer2SoftReset				(Axis:=Screwing2AxisRef, Execute:= TRUE);
		bWarning2						:=	TRUE;			
		udiWarningID					:=	2;	
		IF tonTooLongScrewing2.Q THEN
			sWarningDescription				:=	'Zakręcarka 2 - przekroczenie czasu zakręcania - zmień ust.';
			bWarning2A						:= TRUE;
		END_IF
		IF tonTooLongFinding2.Q THEN
			sWarningDescription				:=	'Zakręcarka 2 - przekroczenie czasu szukania gwintu - zmień ust.';
			bWarning2B						:= TRUE;
		END_IF
		IF tonPosDiff2Error.Q THEN
			sWarningDescription				:=	'Zakręcarka 2 - przekroczenie laga - zmień ust.';
			bWarning2C						:= TRUE;
		END_IF
		IF tonPosTooLowWhenScrewing2.Q THEN
			sWarningDescription				:=	'Zakręcarka 2 - zbyt niska pozycja przy zakrecaniu - zmień ust.';
			bWarning2D						:= TRUE;
		END_IF		
	END_IF


	// Alarm_0460	460	Error	Błąd napędu podnoszenia. Błąd NC: {0}
	//Error 1 - BŁĄD SERWA PODNOSZENIA ZAKRĘCARKI
	IF (HeightAxisRef.Status.Error OR mcHeightMoveAbsolute.Error) AND tonEStop.Q AND NOT bStateError THEN
		arfbAlarm[0].ipArguments.Clear() .AddUDInt(udiHeightServoErrorNr);
		IF NOT arfbAlarm[0].bActive THEN
			mcHeightGearInMultiMaster.Enable	:=	FALSE;
			mcHeightGearOut.Execute				:=	TRUE;		
			arfbAlarm[0].Raise(nTimeStamp:=0);
		END_IF
	ELSE	
		IF  arfbAlarm[0].bActive AND bReset THEN
			arfbAlarm[0].Clear(nTimeStamp:=0, bResetConfirmation:= FALSE);
		END_IF
// 		mcHeightGearInMultiMaster.Enable	:=	FALSE;
// 		mcHeightGearOut.Execute				:=	TRUE;				
// 		bError 								:=	TRUE;
// 		udiErrorID							:=	291;
// 		//udiErrorID 							:=	udiErrorID+iStationIndex;
// 		udiHeightServoErrorNr				:=	HeightAxisRef.Status.ErrorID;
// 		sErrorDescription					:=	'Błąd napędu podnoszenia. Błąd NC:';
// 		sErrorDescription2					:=	F_AxErrMsg(udiHeightServoErrorNr);
	END_IF;
	// Alarm_0461	461	Error	Błąd napędu zakręcającego 1. Błąd NC: {0}
	//Error 2 - BŁĄD SERWA ZAKRĘCAJĄCEGO 1
	IF (Screwing1AxisRef.Status.Error OR mcScrewer1Stop.Error) AND tonEStop.Q AND bEnable1 THEN
		arfbAlarm[1].ipArguments.Clear() .AddUDInt(udiScrewing1ServoErrorNr);
		IF NOT arfbAlarm[1].bActive THEN	
			arfbAlarm[1].Raise(nTimeStamp:=0);
		END_IF
	ELSE	
		IF  arfbAlarm[1].bActive AND bReset THEN
			arfbAlarm[1].Clear(nTimeStamp:=0, bResetConfirmation:= FALSE);
		END_IF
// 		bError 							:=	TRUE;
// 		udiErrorID						:=	292;
// 		//udiErrorID 						:=	udiErrorID+iStationIndex;
// 		udiScrewing1ServoErrorNr		:=	Screwing1AxisRef.Status.ErrorID;
// 		sErrorDescription				:=	'Błąd napędu zakręcającego 1. Błąd NC:';
// 		sErrorDescription2				:=	F_AxErrMsg(udiScrewing1ServoErrorNr);
	END_IF;
	// Alarm_0462	462	Error	Błąd napędu zakręcającego 2. Błąd NC: {0}
	//Error 3 - BŁĄD SERWA ZAKRĘCAJĄCEGO 2
	IF (Screwing2AxisRef.Status.Error OR mcScrewer2Stop.Error) AND tonEStop.Q AND bEnable2 THEN
		arfbAlarm[2].ipArguments.Clear() .AddUDInt(udiScrewing2ServoErrorNr);
		IF NOT arfbAlarm[2].bActive THEN
			iTestError4 := iTestError4 +1;		
			arfbAlarm[2].Raise(nTimeStamp:=0);
		END_IF
	ELSE	
		IF  arfbAlarm[2].bActive AND bReset THEN
			arfbAlarm[2].Clear(nTimeStamp:=0, bResetConfirmation:= FALSE);
		END_IF
// 		bError 							:=	TRUE;
// 		udiErrorID						:=	293;
// 		//udiErrorID 						:=	udiErrorID+iStationIndex;
// 		udiScrewing2ServoErrorNr		:=	Screwing2AxisRef.Status.ErrorID;
// 		sErrorDescription				:=	'Błąd napędu zakręcającego 2. Błąd NC:';
// 		sErrorDescription2				:=	F_AxErrMsg(udiScrewing1ServoErrorNr);
// 		iTestError4 := iTestError4 +1;
	END_IF;
	// Alarm_0463	463	Error	Wartość zadana wysokości jest większa od maksymalnej - zmień ustawienia w recepturze {0}
	//Error 4 - BŁĄD NASTAW MAX
	tonMaxHeight(IN:=(lrHeightReadyPosition>lrMaxHeightPosition OR lrHeightPushingPosition>lrMaxHeightPosition OR lrHeightEndScrewingPosition>lrMaxHeightPosition AND bHomingDone
	AND eState=E_Station.eReady),PT:=T#30S);
	IF tonMaxHeight.Q THEN
		arfbAlarm[3].ipArguments.Clear() .AddLReal(lrMaxHeightPosition);
		IF NOT arfbAlarm[3].bActive THEN		
			arfbAlarm[3].Raise(nTimeStamp:=0);
		END_IF
	ELSE	
		IF  arfbAlarm[3].bActive AND bReset THEN
			arfbAlarm[3].Clear(nTimeStamp:=0, bResetConfirmation:= FALSE);
		END_IF
// 		bError							:=	TRUE;
// 		udiErrorID						:=	294;
// 		//udiErrorID 						:=	udiErrorID+iStationIndex;
// 		sErrorDescription				:=	'Wartość zadana wysokości jest większa od maksymalnej - zmień ustawienia w recepturze';
// 		sErrorDescription2				:=	REAL_TO_STRING(LREAL_TO_INT(lrMaxHeightPosition));
	END_IF
	// Alarm_0464	464	Error	Wartość zadana wysokości jest mniejsza od minimalnej - zmień ustawienia w recepturze {0}
	//Error 5 - BŁAD POZYCJI MINIMALNEJ PODNOŚNIKA 
	IF mcHeightMoveAbsolute.Execute AND mcHeightMoveAbsolute.Position<=lrMinHeightPosition THEN
		arfbAlarm[4].ipArguments.Clear() .AddLReal(lrMinHeightPosition);
		IF NOT arfbAlarm[4].bActive THEN
			mcHeightMoveAbsolute.Execute	:=	FALSE;
			mcHeightStop.Execute			:=	TRUE;			
			arfbAlarm[4].Raise(nTimeStamp:=0);
		END_IF
		IF arfbAlarm[4].bActive AND breset THEN
			fbHeightHardReset						(Execute:=NOT mcHeightMoveAbsolute.Execute,	Axis:=HeightAxisRef);
			mcHeightSoftReset						(Execute:=TRUE,								Axis:=HeightAxisRef);																		
			IF NOT fbHeightHardReset.Busy AND NOT mcHeightSoftReset.Busy AND mcHeightPower.Status AND NOT HeightAxisRef.Status.Error THEN
				fbHeightHardReset					(Execute:=FALSE,							Axis:=HeightAxisRef);
				mcHeightSoftReset					(Execute:=FALSE,							Axis:=HeightAxisRef);
				mcHeightMoveAbsolute.Velocity		:=	lrHeightSpeed;
				mcHeightMoveAbsolute.Position		:=	lrHeightReadyPosition; 
				mcHeightMoveAbsolute.Execute		:=	TRUE;
				IF mcHeightMoveAbsolute.Done THEN
					mcHeightMoveAbsolute.Execute	:=	FALSE;
					mcHeightPower.Override			:=	100;
					mcScrewing1Power.Override		:=	100;
					mcScrewing2Power.Override		:=	100;
					bError							:=	FALSE;
					udiHeightServoErrorNr			:=	0;
					sErrorDescription				:=	'';	
					udiErrorID						:=	0;	
				END_IF
			ELSIF NOT fbHeightHardReset.Busy AND NOT mcHeightSoftReset.Busy AND NOT mcHeightPower.Status AND NOT HeightAxisRef.Status.Error  THEN
				fbHeightHardReset					(Execute:=FALSE,							Axis:=HeightAxisRef);
				mcHeightSoftReset					(Execute:=FALSE,							Axis:=HeightAxisRef);
				mcHeightPower.Override				:=	100;
				mcScrewing1Power.Override			:=	100;
				mcScrewing2Power.Override			:=	100;
				bError 								:=	FALSE;
				udiHeightServoErrorNr				:=	0;
				sErrorDescription					:=	'';	
				udiErrorID							:=	0;	
				arfbAlarm[4].Clear(nTimeStamp:=0, bResetConfirmation:= FALSE);	  	
			END_IF
		END_IF
		
 	ELSE	
 		IF  arfbAlarm[4].bActive AND bReset THEN
 			arfbAlarm[4].Clear(nTimeStamp:=0, bResetConfirmation:= FALSE);
 		END_IF
		
// 		mcHeightMoveAbsolute.Execute	:=	FALSE;
// 		mcHeightStop.Execute			:=	TRUE;	
// 		bError							:=	TRUE;
// 		udiErrorID						:=	295;
// 		//udiErrorID						:=	udiErrorID+iStationIndex;
// 		sErrorDescription				:=	'Wartość zadana wysokości jest mniejsza od minimalnej - zmień ustawienia w recepturze';
// 		sErrorDescription2				:=	LREAL_TO_STRING(lrMinHeightPosition);

	END_IF
	// Alarm_0465	465	Error	Zbyt wysoka temperatura napędu zakręcającego 1 > 130C - zmniejsz moment zakręcania
	//Error 6 - ZBYT WYSOKA TEMPERATURA SILNIKA ZAKRECAJĄCEGO 1
	tonActualMotor1TemperatureTooHigh	(IN:=rActualMotor1Temperature>130, PT:=T#10S);
	IF tonActualMotor1TemperatureTooHigh.Q THEN
		arfbAlarm[5].ipArguments.Clear() .AddLReal(rActualMotor1Temperature);
		IF NOT arfbAlarm[5].bActive THEN		
			arfbAlarm[5].Raise(nTimeStamp:=0);
		END_IF
	ELSE	
		IF  arfbAlarm[5].bActive AND bReset THEN
			arfbAlarm[5].Clear(nTimeStamp:=0, bResetConfirmation:= FALSE);
		END_IF
// 		bError 							:=	TRUE;
// 		udiErrorID						:=	296;
// 		//udiErrorID						:=	udiErrorID+iStationIndex;
// 		sErrorDescription				:=	'Zbyt wysoka temperatura napędu zakręcającego 1 > 130C - zmniejsz moment zakręcania';
// 		sErrorDescription2				:=	INT_TO_STRING(REAL_TO_INT(rActualMotor1Temperature));;
	END_IF
	// Alarm_0466	466	Error	Zbyt wysoka temperatura napędu zakręcającego 2 > 130C - zmniejsz moment zakręcania
	//Error 7 - ZBYT WYSOKA TEMPERATURA SILNIKA ZAKRECAJĄCEGO 2
	tonActualMotor2TemperatureTooHigh	(IN:=rActualMotor2Temperature>130, PT:=T#10S);
	IF tonActualMotor2TemperatureTooHigh.Q THEN
		arfbAlarm[6].ipArguments.Clear() .AddLReal(rActualMotor2Temperature);
		IF NOT arfbAlarm[6].bActive THEN		
			arfbAlarm[6].Raise(nTimeStamp:=0);
		END_IF
	ELSE	
		IF  arfbAlarm[6].bActive AND bReset THEN
			arfbAlarm[6].Clear(nTimeStamp:=0, bResetConfirmation:= FALSE);
		END_IF
// 		bError 							:=	TRUE;
// 		udiErrorID						:=	297;
// 		//udiErrorID						:=	udiErrorID+iStationIndex;
// 		sErrorDescription				:=	'Zbyt wysoka temperatura napędu zakręcającego 2 > 130C - zmniejsz moment zakręcania';
// 		sErrorDescription2				:=	INT_TO_STRING(REAL_TO_INT(rActualMotor1Temperature));;
	END_IF

ELSE
	bError := FALSE;
END_IF


//******************PRZEJŚCIE DO eERROR*****************************

IF bError AND NOT bStateError THEN
	IF eLastState = eRunning THEN
		bCycleNotDone1 := TRUE;
		bCycleNotDone2 := TRUE;		
	END_IF
	eState := E_Station.eError;
END_IF

//****************WYŚWIETLANIE STATUSU BLEDU***********************

(*Wyświetlanie błedu na wyjściu*)
bError							:= FALSE;
FOR nAlarmNumerator := 0 TO 19 DO
	bError						:= bError OR arfbAlarm[nAlarmNumerator].bActive;
END_FOR

(*Przepisywanie nazwy stacji*)
sErrorStationName := WSTRING_TO_STRING(sStationName);

(*Kasowanie casów resettingu*)
//IF  udiErrorID-iStationIndex <>3 THEN
//	iErrorResseting3	:=	0;
//END_IF
END_ACTION

ACTION HeightControlBlocks:
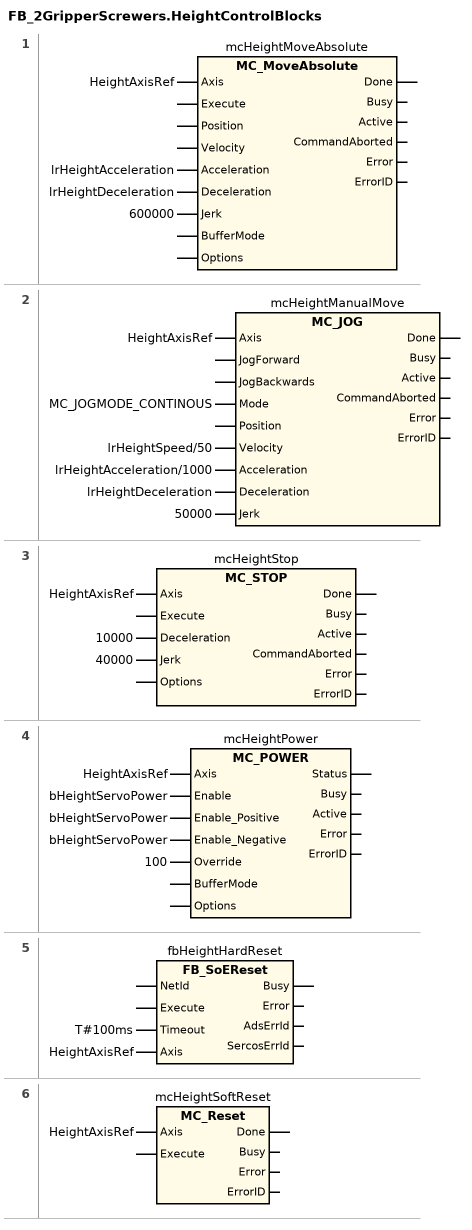
// NETWORK 1
mcHeightMoveAbsolute(
    Axis := HeightAxisRef,
    Acceleration := lrHeightAcceleration,
    Deceleration := lrHeightDeceleration,
    Jerk := 600000); // MC_MoveAbsolute

// NETWORK 2
mcHeightManualMove(
    Axis := HeightAxisRef,
    Mode := MC_JOGMODE_CONTINOUS,
    Velocity := lrHeightSpeed/50,
    Acceleration := lrHeightAcceleration/1000,
    Deceleration := lrHeightDeceleration,
    Jerk := 50000); // MC_JOG

// NETWORK 3
mcHeightStop(Axis := HeightAxisRef, Deceleration := 10000, Jerk := 40000); // MC_STOP

// NETWORK 4
mcHeightPower(
    Axis := HeightAxisRef,
    Enable := bHeightServoPower,
    Enable_Positive := bHeightServoPower,
    Enable_Negative := bHeightServoPower,
    Override := 100); // MC_POWER

// NETWORK 5
fbHeightHardReset(Timeout := T#100ms, Axis := HeightAxisRef); // FB_SoEReset

// NETWORK 6
mcHeightSoftReset(Axis := HeightAxisRef); // MC_Reset

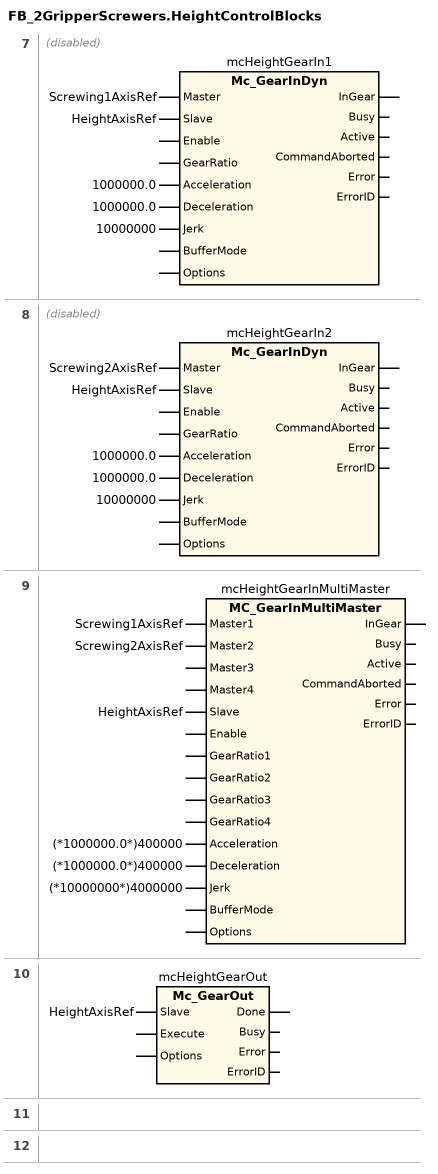
// NETWORK 7 (disabled)
// mcHeightGearIn1(
//     Master := Screwing1AxisRef,
//     Slave := HeightAxisRef,
//     Acceleration := 1000000.0,
//     Deceleration := 1000000.0,
//     Jerk := 10000000); // Mc_GearInDyn

// NETWORK 8 (disabled)
// mcHeightGearIn2(
//     Master := Screwing2AxisRef,
//     Slave := HeightAxisRef,
//     Acceleration := 1000000.0,
//     Deceleration := 1000000.0,
//     Jerk := 10000000); // Mc_GearInDyn

// NETWORK 9
mcHeightGearInMultiMaster(
    Master1 := Screwing1AxisRef,
    Master2 := Screwing2AxisRef,
    Slave := HeightAxisRef,
    Acceleration := (*1000000.0*)400000,
    Deceleration := (*1000000.0*)400000,
    Jerk := (*10000000*)4000000); // MC_GearInMultiMaster

// NETWORK 10
mcHeightGearOut(Slave := HeightAxisRef); // Mc_GearOut

// NETWORK 11

// NETWORK 12
END_ACTION

ACTION Homing:
//BAZOWANIE 
bGripper1Actuator					:= FALSE;
bGripper2Actuator 					:= FALSE;
//Wylaczanie serwa zakręcania podczas bazowania
mcScrewing1Power.Override			:=	100;
//mcScrewer1Stop.Execute				:=	bEnable1;
mcScrewer1MoveVelocity.Execute		:=	FALSE;
mcScrewer1MoveVelocity2.Execute		:=	FALSE;
mcScrewer1MoveVelocity3.Execute		:=	FALSE;
mcScrewer1ManualMove.JogBackwards	:=	FALSE;
mcScrewer1ManualMove.JogForward		:=	FALSE;

mcScrewing2Power.Override			:=	100;
//mcScrewer2Stop.Execute				:=	bEnable2;
mcScrewer2MoveVelocity.Execute		:=	FALSE;
mcScrewer2MoveVelocity2.Execute		:=	FALSE;
mcScrewer2MoveVelocity3.Execute		:=	FALSE;
mcScrewer2ManualMove.JogBackwards	:=	FALSE;
mcScrewer2ManualMove.JogForward		:=	FALSE;

bHeightServoPower					:=	TRUE;
	
IF mcHeightPower.Status THEN
		
	IF bHoming THEN // Bazowanie - podjazd do góry i ustawienie obrotu
		CASE iHomingCase OF
		
			0:
				iHomingCase							:= iHomingCase	+	10;
				
			10:	//Podjazd do góry
				mcHeightMoveAbsolute.Velocity		:=	100;
				mcHeightMoveAbsolute.Position		:=	lrMaxHeightPosition;
				mcHeightMoveAbsolute.Execute		:=	TRUE;
				mcHeightPower.Override				:=	100;
				mcScrewing1Power.Override			:=	100;
				mcScrewing2Power.Override			:=	100;
				IF mcHeightMoveAbsolute.Done THEN
					mcHeightMoveAbsolute.Execute	:=	FALSE;
					iHomingCase						:= iHomingCase	+	10;					
				END_IF
				
			20: //Obrót 1
				IF 		M_PrepareToReady(	AxisRef			:=  Screwing1AxisRef,	(*Obrót*) 		
											iGripperArms	:=	2					)			OR NOT bEnable1
				THEN
					iHomingCase						:= iHomingCase	+	10;	
				END_IF
			
			30: //Obrót 2
				IF 		M_PrepareToReady(	AxisRef			:=  Screwing2AxisRef,	(*Obrót*) 		
											iGripperArms	:=	2					)			OR NOT bEnable2
				THEN
					iHomingCase						:= iHomingCase	+	10;	
				END_IF
			
			40:	//Koniec
				eState								:= E_Station.eHomingDone;
				iHomingCase							:= 0;
		END_CASE
	END_IF
	IF bHeightSet THEN // Ustawianie wysokości zadanej z receptury - uważać na kolizje
		mcHeightManualMove.Acceleration				:=  lrHeightAcceleration;
		mcHeightManualMove.Deceleration				:=  lrHeightDeceleration;		
		mcHeightManualMove.Velocity					:=  lrHeightSpeed;
		mcHeightManualMove.JogForward				:=	HeightAxisRef.NcToPlc.ActPos<=lrHeightReadyPosition AND HeightAxisRef.NcToPlc.ActPos<=lrMaxHeightPosition;
		mcHeightManualMove.JogBackwards				:=	HeightAxisRef.NcToPlc.ActPos>=lrHeightReadyPosition AND HeightAxisRef.NcToPlc.ActPos>=lrMinHeightPosition;
		IF ABS(HeightAxisRef.NcToPlc.ActPos-lrHeightReadyPosition)<1 THEN
			mcHeightManualMove.JogForward			:=	FALSE;
			mcHeightManualMove.JogBackwards			:=	FALSE;
			eState									:=	E_Station.eHomingDone;
		END_IF
			bHeighSetNotDone						:=	TRUE;		
	END_IF		
END_IF
END_ACTION

ACTION Limits:
(*Wywowyłanie na początku*)

(*Prędkość zakręcania*)
IF lrScrewerSpeed > lrMaxScrewerSpeed 	THEN		lrScrewerSpeed	:= lrMaxScrewerSpeed;				END_IF
IF lrScrewerSpeed = 0 					THEN		lrScrewerSpeed	:= lrMaxScrewerSpeed/2;				END_IF

(*Parametry gwintu*)
IF lrPackageTurnoversToFullScrewed < 0.1	THEN		lrPackageTurnoversToFullScrewed := 0.1;			END_IF
IF lrPackageThreadPitch < 0.5 				THEN		lrPackageThreadPitch := 0.5;					END_IF
IF lrPackageThreadTimes < 1 				THEN		lrPackageThreadTimes := 1;						END_IF

(*Pozycje*)
IF lrHeightReadyPosition		< 10		THEN		lrHeightReadyPosition		:=	lrMaxHeightPosition - 5;		END_IF
IF lrHeightPushingPosition		< 10		THEN		lrHeightPushingPosition		:=	lrMaxHeightPosition - 10;		END_IF
IF lrHeightEndScrewingPosition	< 10		THEN	    lrHeightEndScrewingPosition	:=	lrMaxHeightPosition - 10;		END_IF

(*Override*)
IF lrManualOverride < 10 					THEN		lrManualOverride	:= 10;						END_IF


(*Inny parametr*)
//...
END_ACTION

(*
Obrót chwytaka o określony kąt, tak żeby 
był zawsze skeirowany w tą samą stronę
Instrukcja:
- włączyć w drivie Scaling->Modulo data storage source - Feeback 1
- ustawić drive Scaling->position offset setting 0 stopni na odpowiedniej pozycji na enkoderze
- wgrać z drive Save NC parameters
- w drivie jeszcze raz ustawić parametr na 359?	
*)

METHOD M_PrepareToReady : BOOL

VAR_INPUT
	iGripperArms	:	INT;			//Ilość ramieni chwytaka (domyślnie 2)
END_VAR
VAR_IN_OUT
	AxisRef			:	AXIS_REF;
END_VAR
VAR
	lrAxisRefActPos: LREAL;
	lrDivider: LREAL;

END_VAR
(*Przypisania dla ułatwienia*)
lrAxisRefActPos := AxisRef.NcToPlc.ActPos;
lrDivider		:= 360.0/iGripperArms;

CASE iMStep OF
	
	0: // Czy tu nie trzeba zrobić 
		iMStep							:= iMStep + 10;
		
	10: // Obliczanie najkrótszej pozycji, zależnie od ilość ramion chwytaka
		uiScrewing1TorqueControl		:= 6000; // Ustawianie momentu bo moze byc 0
		uiScrewing2TorqueControl		:= 6000; // Ustawianie momentu bo moze byc 0
	
	
	IF lrAxisRefActPos	>	0 THEN 	//Jeżeli aktualna pozycja jest >0 //w
		IF LMOD(lrAxisRefActPos,lrDivider)>(lrDivider/2) THEN // Dobieranie pozycji, tak żeby było bliżej
			mcMoveAbsolute.Position		:=	lrAxisRefActPos+lrDivider			-	LMOD(lrAxisRefActPos,lrDivider);
		ELSE
			mcMoveAbsolute.Position		:=	lrAxisRefActPos+lrDivider			-	LMOD(lrAxisRefActPos,lrDivider);
			//mcMoveAbsolute.Position	:=	lrAxisRefActPos						-	LMOD(lrAxisRefActPos,lrDivider);			
		END_IF
	ELSE 							//Jezeli aktualna mniejsza od 0
		IF LMOD(ABS(lrAxisRefActPos),lrDivider)>(lrDivider/2) THEN // Dobieranie pozycji, tak żeby było bliżej
			mcMoveAbsolute.Position		:=	lrAxisRefActPos-lrDivider			-	LMOD(lrAxisRefActPos,lrDivider);
		ELSE
			mcMoveAbsolute.Position		:=	lrAxisRefActPos-lrDivider			-	LMOD(lrAxisRefActPos,lrDivider);
			//mcMoveAbsolute.Position	:=	lrAxisRefActPos						-	LMOD(lrAxisRefActPos,lrDivider);{warning 'wył obrot'}		
		END_IF
	END_IF
		iMStep						:= iMStep + 10;

	20: //Ruch
		mcMoveAbsolute.Execute		:=	TRUE;
		iMStep						:= iMStep + 10;	
	
	30: //Wykonano
		IF mcMoveAbsolute.Done THEN
			mcMoveAbsolute.Execute	:=	FALSE;
			iMStep					:= 100;			
		END_IF
		
	100: //Koniec
		M_PrepareToReady				:= TRUE;
		iMStep						:= 0;
	
END_CASE


mcMoveAbsolute(
	Axis:= AxisRef, 
	Execute:= , 
	Position:= , 
	Velocity:= 		4000, 
	Acceleration:=	24000, 
	Deceleration:=	24000, 
	Jerk:= 			10000000, 
	BufferMode:= , 
	Options:= , 
	Done=> , 
	Busy=> , 
	Active=> , 
	CommandAborted=> , 
	Error=> , 
	ErrorID=> );
END_METHOD

ACTION ManualMovements:
//W trybie ruchów manualnych wykonuj ruchy za pomocą rozkazów manualnych
IF NOT bRun1 AND NOT bRun2 AND NOT bAdjustingTorque THEN
	mcHeightPower.Override				:=	lrManualOverride;
	mcScrewing1Power.Override			:=	lrManualOverride;
	mcScrewing2Power.Override			:=	lrManualOverride;
	uiScrewing1TorqueControl			:=	(INT_TO_UINT(iScrewer1SetTorque+5)*10)*BOOL_TO_UINT(bManualScrew1Clockwise OR bManualScrew1CClockwise);
	uiScrewing2TorqueControl			:=	(INT_TO_UINT(iScrewer2SetTorque+5)*10)*BOOL_TO_UINT(bManualScrew2Clockwise OR bManualScrew2CClockwise);
	mcHeightManualMove.JogForward		:=	bManualHeightUp;
	mcHeightManualMove.JogBackwards		:=	bManualHeightDown;
	mcScrewer1ManualMove.JogForward		:=	bManualScrew1Clockwise;
	mcScrewer1ManualMove.JogBackwards	:=	bManualScrew1CClockwise;
	mcScrewer2ManualMove.JogForward		:=	bManualScrew2Clockwise;
	mcScrewer2ManualMove.JogBackwards	:=	bManualScrew2CClockwise;
	bGripper1Actuator					:=	bManualGripper1;
	bGripper2Actuator					:=	bManualGripper2;	
ELSE	//Kasuje zeby po cyklu nic sie nie poruszało
	bManualGripper1						:= FALSE;
	bManualGripper2 					:= FALSE;
END_IF


IF bHoming OR bHeightSet THEN
	eState:=E_Station.eHoming;
END_IF
	
IF NOT bAdjustingTorque THEN
	Running();
END_IF

IF NOT bRun1 AND NOT bRun2 THEN
	bCycleDone1 				:= FALSE;
	bCycleNotDone1 				:= FALSE;	
	bCycleDone2					:= FALSE;
	bCycleNotDone2 				:= FALSE;	
	bWarning1					:= FALSE;	
	bWarning2					:= FALSE;	
END_IF
END_ACTION

ACTION ManualMovementsStepMode:
bManualHeightUp;
bManualHeightDown;
bStepMode;		
lrSetPosStepMode;

// Limity
IF lrSetPosStepMode < 1			THEN	lrSetPosStepMode := 1;	END_IF
IF lrSetPosStepMode > 10		THEN	lrSetPosStepMode := 10;	END_IF

// Zabezpieczenie przed zbyt szybkim włączaniem
tofStepModeMoving				(IN := bStepModeMoving,					PT:=T#500MS);

// Możliwe włączenie jeżeli zakończyło poprzedni ruch
rtStepModeUp					(CLK :=	bStepMode AND NOT tofStepModeMoving.Q	AND bManualHeightUp,	Q=>);
rtStepModeDown					(CLK :=	bStepMode AND NOT tofStepModeMoving.Q 	AND bManualHeightDown,	Q=>);

// Włączenie ruchu w górę
IF rtStepModeUp.Q THEN
	bStepModeMoving				:= TRUE;
	lrStepModeHeightMotorSV		:= HeightAxisRef.NcToPlc.ActPos	+	lrSetPosStepMode;
END_IF

// Włączenie ruchu w dół
IF rtStepModeDown.Q THEN
	bStepModeMoving				:= TRUE;
	lrStepModeHeightMotorSV		:= HeightAxisRef.NcToPlc.ActPos	-	lrSetPosStepMode;
END_IF
// DODAĆ RESET bStepModeMoving PO BLEDZIE!
// Ruch w górę !SPRAWDZIC ZNAKI!
IF bStepModeMoving THEN
	mcHeightManualMove.JogForward		:=	HeightAxisRef.NcToPlc.ActPos	<=	lrStepModeHeightMotorSV;
	mcHeightManualMove.JogBackwards		:=	HeightAxisRef.NcToPlc.ActPos	>=	lrStepModeHeightMotorSV;	
	
	IF ABS(HeightAxisRef.NcToPlc.ActPos-lrStepModeHeightMotorSV) < 0.5	OR	// Pozycja osiągnięta (co do 1mm)
			(HeightAxisRef.NcToPlc.ActPos-iToolHeight<=lrMinHeightPosition)					OR 	// Pozycja poniżej minimalnej
			(HeightAxisRef.NcToPlc.ActPos>=lrMaxHeightPosition) 					// Pozycja powyżej maksymalnej
	THEN
		mcHeightManualMove.JogForward	:= FALSE;
		mcHeightManualMove.JogForward	:= FALSE;
		bStepModeMoving					:= FALSE;
		bManualHeightUp					:= FALSE;
		bManualHeightDown				:= FALSE;
	END_IF	
END_IF
END_ACTION

ACTION ReadScrewingTorque:
//Zapisywanie momentu w trakcie zakręcania
//IF eRunningState = E_GripperScrewer.eScrewing OR  eRunningState = E_GripperScrewer.eHolding THEN
	//Zapisywanie maksymalnego momentu zakręcania 1
IF ABS(ABS(lrStartPosition1)-ABS(Screwing1AxisRef.NcToPlc.ActPos))>(lrPackageTurnoversToFullScrewed*360.0/6) AND 
		tonMomentaryScrewing1Timer.IN  OR (tonTightScrewing1Timer.IN AND NOT bOptionMomentaryMode)
THEN //Zapisywanie momentu bez tego zwiększonego przy uruchomieniu

	IF (ABS(lrScrewer1ActualTorque))/100.0*1.5  > lrScrewer1TorqueCV THEN 
		lrScrewer1TorqueCV := (ABS(lrScrewer1ActualTorque))/100.0*1.5; 
	END_IF
END_IF
	//Zapisywanie maksymalnego momentu zakręcania 2
IF ABS(ABS(lrStartPosition2)-ABS(Screwing2AxisRef.NcToPlc.ActPos))>(lrPackageTurnoversToFullScrewed*360.0/6) AND 
		tonMomentaryScrewing2Timer.IN OR (tonTightScrewing2Timer.IN AND NOT bOptionMomentaryMode) 
THEN //Zapisywanie momentu bez tego zwiększonego przy uruchomieniu
	IF ABS(lrScrewer2ActualTorque)/100.0*1.5 > lrScrewer2TorqueCV THEN 
		lrScrewer2TorqueCV := (ABS(lrScrewer2ActualTorque))/100.0*1.5; 
	END_IF
END_IF
//END_IF
//Kasowanie na starcie
rtRun1(CLK:=bRun1, Q=>);
rtRun2(CLK:=bRun2, Q=>);
IF rtRun1.Q THEN
	lrScrewer1TorqueCV	:= 	0;
END_IF
IF rtRun2.Q THEN
	lrScrewer2TorqueCV	:=	0;
END_IF
END_ACTION

ACTION ResetCommands:
iCloseGripperBeforeScrewingCASE			:=	0;
iScrewingCase							:= 0;
iStoppingCase 							:= 0;
iGoingUpCase							:= 0;
iHomingCase								:= 0;
iPreparingToReadyCase					:= 0;
iToPushingPositionCase					:= 0;
iMStep									:= 0;

iErrorResseting3					:= 0;

mcHeightGearInMultiMaster.Enable	:=	FALSE;
mcHeightGearOut.Execute				:=	FALSE;
mcHeightMoveAbsolute.Execute		:=	FALSE;
mcHeightStop.Execute				:=	FALSE;
mcHeightManualMove.JogBackwards		:=	FALSE;
mcHeightManualMove.JogForward		:=	FALSE;
mcHeightSoftReset					(Execute:=FALSE,Axis:=HeightAxisRef);
fbHeightHardReset					(Execute:=FALSE,Axis:=HeightAxisRef);

mcMoveAbsolute.Execute				:=	FALSE;			
mcScrewer1Stop.Execute				:=	FALSE;
mcScrewer2Stop.Execute				:=	FALSE;
mcScrewer1ManualMove.JogBackwards	:=	FALSE;
mcScrewer1ManualMove.JogForward		:=	FALSE;
mcScrewer2ManualMove.JogBackwards	:=	FALSE;
mcScrewer2ManualMove.JogForward		:=	FALSE;
mcScrewer1MoveVelocity.Execute		:=	FALSE;
mcScrewer2MoveVelocity.Execute		:=	FALSE;
mcScrewer1MoveVelocity2.Execute		:=	FALSE;
mcScrewer2MoveVelocity2.Execute		:=	FALSE;
mcScrewer1MoveVelocity3.Execute		:=	FALSE;
mcScrewer2MoveVelocity3.Execute		:=	FALSE;
mcScrewer1TorqueControl.Execute		:=	FALSE;
mcScrewer2TorqueControl.Execute		:=	FALSE;
mcScrewer1MoveAbsolute.Execute		:=	FALSE;
mcScrewer2MoveAbsolute.Execute		:=	FALSE;


bStepModeMoving						:=	FALSE;
mcScrewer1SoftReset					(Execute:=FALSE,Axis:=Screwing1AxisRef);	
mcScrewer2SoftReset					(Execute:=FALSE,Axis:=Screwing2AxisRef);	
fbScrewer1HardReset					(Execute:=FALSE,Axis:=Screwing1AxisRef);	
fbScrewer2HardReset					(Execute:=FALSE,Axis:=Screwing2AxisRef);	


bGripper1Actuator					:=	FALSE;
bGripper2Actuator					:=	FALSE;
END_ACTION

ACTION Running:
tonFindingScrew		(IN:=eRunningState= E_GripperScrewer.eFindingScrew, PT:=T#80MS);
tonScrew1Found		(IN:=bScrew1Found,									PT:=T#50MS);
tonScrew2Found		(IN:=bScrew2Found,									PT:=T#50MS);

CASE eRunningState OF

//====================================
	
	(*Oczekiwanie na wykonanie pojedynczego cyklu*)
	E_GripperScrewer.eReady:
	
        mcScrewer1SoftReset								(Axis:=Screwing1AxisRef, Execute:=FALSE);                                       	
		mcScrewer1MoveVelocity.Execute					:=	FALSE;
		mcScrewer1MoveVelocity2.Execute					:=	FALSE;
		mcScrewer1MoveVelocity3.Execute					:=	FALSE;		
		uiScrewing1TorqueControl						:=	6000;
        mcScrewer2SoftReset								(Axis:=Screwing1AxisRef, Execute:=FALSE);                                       	
		mcScrewer2MoveVelocity.Execute					:=	FALSE;
		mcScrewer2MoveVelocity2.Execute					:=	FALSE;
		mcScrewer2MoveVelocity3.Execute					:=	FALSE;		
		uiScrewing2TorqueControl						:=	6000;		
		mcHeightMoveAbsolute.Execute					:=	FALSE;
		uiHeightTorqueControl							:=	6000;                                      	

		bScrewed1										:=	FALSE;
		bScrewed2										:=	FALSE;
		bScrew1Found									:=	FALSE;
		bScrew2Found									:=	FALSE;		
 		                                       	
		IF NOT bCycleDone1 AND NOT bCycleNotDone1 AND NOT bCycleDone2 AND NOT bCycleNotDone2 THEN                                           	
			IF bRun1 OR bRun2 THEN                	
				mcHeightMoveAbsolute.Execute			:=	FALSE;				
				IF lrHeightEndScrewingPosition = lrHeightPushingPosition THEN
					eRunningState						:=	E_GripperScrewer.eToScrewingPosition;
				ELSE
					eRunningState						:=	E_GripperScrewer.eToPushingPosition;	
				END_IF	
			END_IF
		END_IF
		
//====================================		
	(*Ruch na pozycję wbijania*)			
	E_GripperScrewer.eToPushingPosition:
	
		Running2ToPushingPosition();

//====================================					
	(*Ruch na pozycję zakręcania*)		
	E_GripperScrewer.eToScrewingPosition:
	
		mcScrewer1MoveVelocity.Velocity					:=	lrScrewerSpeed;
		mcScrewer2MoveVelocity.Velocity					:=	lrScrewerSpeed;
		mcHeightMoveAbsolute.Position					:=	lrHeightEndScrewingPosition;
		mcHeightMoveAbsolute.Velocity					:=	lrHeightSpeed;
		mcHeightMoveAbsolute.Execute					:=	NOT mcHeightMoveAbsolute.Done;
		//Jeśli zakręcarka na wysokości zakręcania przejdź do stanu zakręcania
		IF mcHeightMoveAbsolute.Done AND 
			(mcScrewer1MoveRelative.Done OR NOT mcScrewer1MoveRelative.Execute OR NOT bRun1 OR NOT bOptionFindScrewRotateFromPushingToScrewingSensor OR  bOptionCapPositioning) AND  //bOptionCapPositioning?
			(mcScrewer2MoveRelative.Done OR NOT mcScrewer2MoveRelative.Execute OR NOT bRun2 OR NOT bOptionFindScrewRotateFromPushingToScrewingSensor OR  bOptionCapPositioning) 
			
		THEN
			mcScrewer1MoveRelative.Execute				:= FALSE;
			mcScrewer2MoveRelative.Execute				:= FALSE;
			mcHeightMoveAbsolute.Execute				:=	FALSE;
			
			IF iTool <> 2 THEN
				bGripper1Actuator						:=	bRun1 AND NOT bOptionCapPushingWithoutScrewing;
				bGripper2Actuator						:=	bRun2 AND NOT bOptionCapPushingWithoutScrewing;	
			ELSE
				bGripper1Actuator						:=	FALSE;
				bGripper2Actuator						:=	FALSE;	
			END_IF
			
			IF bOptionFindScrewInScrewingPosition AND NOT bOptionFindScrewInPushingPosition THEN
				IF 	bOptionOpenedGripperWhenFindingScrew THEN //Opcja - szukanie gwintu na otwartym chwytaku
						bGripper1Actuator				:=	FALSE;
						bGripper2Actuator				:=	FALSE;
				END_IF
				IF (tonGripper1Delay.Q OR sTool = 'ksztaltowa/do kulek' OR NOT bRun1) AND (tonGripper2Delay.Q OR sTool = 'ksztaltowa/do kulek' OR NOT bRun2) OR bOptionOpenedGripperWhenFindingScrew THEN
					iFindingScrewCASE					:=	0;
					eRunningState						:=	E_GripperScrewer.eFindingScrew;
				END_IF
				uiScrewing1TorqueControl				:=	6000; //Tutaj na wszelki wypadek żeby przyjeło wartość
				uiScrewing2TorqueControl				:=	6000; //Tutaj na wszelki wypadek żeby przyjeło wartość
			ELSE
				lrStartPosition1:=Screwing1AxisRef.NcToPlc.ActPos;
				lrStartPosition2:=Screwing2AxisRef.NcToPlc.ActPos;		
				IF (tonGripper1Delay.Q OR sTool = 'ksztaltowa/do kulek' OR NOT bRun1) AND (tonGripper2Delay.Q OR sTool = 'ksztaltowa/do kulek' OR NOT bRun2) OR bOptionCapPushingWithoutScrewing THEN
					IF NOT bOptionCapPushingWithoutScrewing THEN (*Opcja bez zakręcania/samo wbijanie*)
						IF NOT bHeightGearingWithScrewer THEN 	(* Wersja bez gearowania*)
							mcScrewer1MoveVelocity.Direction	:=	MC_Positive_Direction;
							mcScrewer1MoveVelocity.Velocity		:=	lrScrewerSpeed;
							mcScrewer1MoveVelocity.Execute		:=	bRun1;
							mcScrewer2MoveVelocity.Direction	:=	MC_Positive_Direction;
							mcScrewer2MoveVelocity.Velocity		:=	lrScrewerSpeed;
							mcScrewer2MoveVelocity.Execute		:=	bRun2;					
							eRunningState						:=	E_GripperScrewer.eScrewing;
						ELSE 									(* Wersja z gearowaniem*)
							eRunningState						:=	E_GripperScrewer.eScrewing;
						END_IF
					ELSE
						eRunningState						:=	E_GripperScrewer.eHolding;
					END_IF
				END_IF
			END_IF
		END_IF
	
//====================================		
			
	(*Szukanie gwintu - jeżeli włączone*)		
	E_GripperScrewer.eFindingScrew:
		
		Running5FindingScrew();

//====================================		
		
	(*Zakręcanie*)
	E_GripperScrewer.eScrewing:

			IF NOT  bHeightGearingWithScrewer THEN 	
				(* Wersja 1 - bez gearowania **********************************************************) 
				mcHeightMoveAbsolute.Position	:=	HeightAxisRef.NcToPlc.ActPos-lrPackageThreadPitch;
				mcHeightMoveAbsolute.Velocity	:=	lrHeightScrewingDistanceSpeed;
				mcHeightMoveAbsolute.Execute	:=	TRUE;				 	  
				mcScrewer1MoveVelocity.Velocity	:=	lrScrewerSpeed;
				mcScrewer2MoveVelocity.Velocity	:=	lrScrewerSpeed;
				
				(*Wymuszanie zwiększonego momentu przez 1/4 całego zakręcania*)
				IF ABS(ABS(lrStartPosition1)-ABS(Screwing1AxisRef.NcToPlc.ActPos))> (lrPackageTurnoversToFullScrewed*360.0/5)  THEN 
					uiScrewing1TorqueControl:=INT_TO_UINT(iScrewer1SetTorque+3)*10;
				ELSE
					uiScrewing1TorqueControl:=(INT_TO_UINT(iScrewer1SetTorque+3)*10)+500;	
				END_IF
				(*Wymuszanie zwiększonego momentu przez 1/4 całego zakręcania*)
				IF ABS(ABS(lrStartPosition2)-ABS(Screwing2AxisRef.NcToPlc.ActPos))>(lrPackageTurnoversToFullScrewed*360.0/5) THEN 
					uiScrewing2TorqueControl:=INT_TO_UINT(iScrewer2SetTorque+3)*10;
				ELSE
					uiScrewing2TorqueControl:=(INT_TO_UINT(iScrewer2SetTorque+3)*10)+500;	
				END_IF
				
				IF tonTightScrewing1Timer.Q OR bWarning1 THEN
					bGripper1Actuator					:=	FALSE;
					mcScrewer1MoveVelocity.Execute		:=	FALSE;
					mcScrewer1SoftReset					(Axis:=Screwing1AxisRef, Execute:= bRun1);
					uiScrewing1TorqueControl			:=	0;
					bScrewed1							:=	TRUE;		
				END_IF
				
				IF tonTightScrewing2Timer.Q OR bWarning2 THEN
					bGripper2Actuator					:=	FALSE;
					mcScrewer2MoveVelocity.Execute		:=	FALSE;
					mcScrewer2SoftReset					(Axis:=Screwing2AxisRef, Execute:= bRun2);
					uiScrewing2TorqueControl			:=	0;
					bScrewed2							:=	TRUE;		
				END_IF
					   
				IF  mcHeightMoveAbsolute.DONE AND (bScrewed1 OR NOT bRun1) AND (bScrewed2 OR NOT bRun2) THEN
					eRunningState						:=	E_GripperScrewer.eHolding;
					mcHeightMoveAbsolute.Execute		:=	FALSE;	 
				END_IF 
				
			ELSE
				(* Wersja 2 - gearowanie *) 
				(*Ustawianie ratio gearowania, musi być poza Casem***********************************)
				// Pobieranie GearRatio z tego obrotu który dłużej zakręca, czyli jeżeli jeden się zatrzyma to pobiera GearRatio z drugiego jeżeli dalej się obraca
				// Oś 1 jest priorytetem, jeżeli się zatrzyma to bieże z drugiego jeżeli dalej sie obraca	
				lrGearRatio1							:= -( (lrPackageThreadPitch*lrPackageThreadTimes) / 360.0 + 0.000000000001);
				lrGearRatio2							:= -( (lrPackageThreadPitch*lrPackageThreadTimes) / 360.0 + 0.000000000001);
				
				IF NOT bOptionMomentaryMode THEN
					lrSf1									:= Screwing1AxisRef.NcToPlc.ActVelo/(mcScrewer1MoveVelocity.Velocity+ 0.000000000001);
					lrSf2									:= Screwing2AxisRef.NcToPlc.ActVelo/(mcScrewer2MoveVelocity.Velocity+ 0.000000000001);	
				ELSE
					lrSf1									:= Screwing1AxisRef.NcToPlc.ActVelo/(Screwing1AxisRef.NcToPlc.SetVelo	+ 0.000000000001);
					lrSf2									:= Screwing2AxisRef.NcToPlc.ActVelo/(Screwing2AxisRef.NcToPlc.SetVelo	+ 0.000000000001);	
					IF Screwing1AxisRef.NcToPlc.ActVelo < 1 OR Screwing1AxisRef.NcToPlc.SetVelo < 1 THEN
						lrSf1	 := 0;
					END_IF
					IF Screwing2AxisRef.NcToPlc.ActVelo < 1 OR Screwing2AxisRef.NcToPlc.SetVelo < 1 THEN
						lrSf2	:=	0;
					END_IF
				END_IF

				
				mcHeightGearInMultiMaster.GearRatio1 	:= lrSf1 * 	lrGearRatio1;				
				mcHeightGearInMultiMaster.GearRatio2 	:= lrSf2 * 	lrGearRatio2;
				
